// TwinCAT 3 PLC project Untitled1
// ProjectVersion: 1.2.0
// ProgramVersion: 3.1.4023.0
// libraries:
//   Tc2_DataExchange, * (Beckhoff Automation GmbH)
//   Tc2_MC2, * (Beckhoff Automation GmbH)
//   Tc2_SerialCom, * (Beckhoff Automation GmbH)
//   Tc2_Standard, * (Beckhoff Automation GmbH)
//   Tc2_System, * (Beckhoff Automation GmbH)
//   Tc2_Utilities, * (Beckhoff Automation GmbH)
//   Tc3_Module, * (Beckhoff Automation GmbH)
// project tree:
//   DUTs/Communication/Axis/ commAxis.TcDUT
//   DUTs/Communication/ Block128Words.TcDUT, CellDataBlock.TcDUT, commManual.TcDUT, contextVacuum.TcDUT, contextManual.TcDUT
//   DUTs/Communication/Command/ commCommandBase.TcDUT, commCommandGeneric.TcDUT, commCommandPos.TcDUT
//   DUTs/Communication/Cylinder/ commCylinder.TcDUT
//   DUTs/Communication/Signal/ commSignal.TcDUT
//   DUTs/Communication/Unit/ commUnit.TcDUT, commUnitConfig.TcDUT, commUnitGeneric.TcDUT, commUnitController.TcDUT
//   DUTs/Definitions/ eAdsIndexGroups.TcDUT, eCommandTypes.TcDUT, eErrorCodes.TcTLEO, eModes.TcDUT, eCategrories.TcDUT, eCylinderCommands.TcDUT, eErrorClearWays.TcDUT, ePositionType.TcDUT, eOperationModes.TcDUT, eSpecialStates.TcDUT
//   DUTs/HRASI/ defAlignment.TcDUT, defHandshake.TcDUT, defItem.TcDUT, eErrorReasons.TcDUT, eSCARATask.TcTLEO, defSensorPair.TcDUT
//   DUTs/Internal/ ParameterGeneric.TcDUT, ParameterSet.TcDUT, ParametersHome.TcPOU, ParametersPosition.TcDUT
//   DUTs/ ioBundleConveyor.TcDUT, ioBundleET.TcDUT, ioBundleLabelGripper.TcDUT, ioBundlePrinterApplicator.TcDUT
//   DUTs/Material/ MaterialBlock.TcDUT, MaterialHeader.TcDUT
//   GVLs/ GVL.TcGVL, GVL_DeivceList.TcGVL
//   / PlcTask.TcTTO
//   POUs/ CheckBounds.TcPOU, CheckPointer.TcPOU, IncNoOverflow.TcPOU, MAIN.TcPOU
//   POUs/Foundation/ CommonBase.TcPOU, ExecuteBase.TcPOU, InterfaceControlV2.TcPOU, InterfaceManualV2.TcPOU, ProgrammedOutput.TcPOU, RunGroupNode.TcPOU, RunMaterial.TcPOU, RunSafetyFacilityProcessor.TcPOU, RunUnitControllerV2.TcPOU, RunUnitSlave.TcPOU, RunVacuum.TcPOU, SemephoreV1.TcPOU, SemephoreV2.TcPOU, RunAxis.TcPOU, InterfaceControlV1.TcPOU, RunCylinder.TcPOU, InterfaceManualV1.TcPOU, RunSignal.TcPOU, RunUnitControllerV1.TcPOU, RunUnitGeneric.TcPOU, RunUnitIndexerMaster.TcPOU, RunUnitTransporterBase.TcPOU
//   POUs/Helper/ CellDataBlock2Parameter.TcPOU, Parameter2CellDataBlock.TcPOU
//   POUs/Stations/CellularD/ RunCableHolder.TcPOU, RunGradeOutput.TcPOU, RunLabelHandler.TcPOU
//   POUs/Stations/HRASI/InitAndTaskControl/ RunCoordinator.TcPOU, RunInitClamperAndIndexer.TcPOU, RunInitScaraAndRack.TcPOU
//   POUs/Stations/HRASI/ RunBin.TcPOU, RunClamper.TcPOU, RunCommonRack.TcPOU, helperOutputSelection.TcPOU, RunAoiInspectionV1.TcPOU, RunBridge.TcPOU, RunDimmerControl.TcPOU, RunLoading.TcPOU, RunPnueIndexer.TcPOU, RunScaraAgent.TcPOU
//   POUs/Stations/ RunAoiHandshaking.TcPOU (excluded from build), RunAxisAoiView.TcPOU (excluded from build), RunAxisInspection.TcPOU (excluded from build), RunBottomView.TcPOU (excluded from build), RunETest.TcPOU (excluded from build), RunInputV1.TcPOU (excluded from build), RunUnitCellularAIO.TcPOU (excluded from build), RunUnitCellularC.TcPOU (excluded from build), RunLifterCelluar.TcPOU (excluded from build), RunUnitCellularA.TcPOU (excluded from build), RunUnitDummy.TcPOU (excluded from build)
// real-time tasks:
//   TASK PlcTask: cycle T#10ms, priority 20, ADS port 350
// motion (NC):
//   TASK NC-Task 1 SAF: cycle T#2ms, priority 4, ADS port 501
//   TASK NC-Task 1 SVB: cycle T#10ms, priority 8, ADS port 511
//   AXIS Simu1 (id 1)
//     OtherSettings: AllowMotionCmdToSlave=true
//     encoder EncType=1
//     drive DrvType=5
//       Analog: ScaleFactorActTorque=0.1
//       TimeComp: TaskDelayCycles=1
//     controller CtrType=1
//       CtrPara: PriorControlFactor=1
//         Observer: BandWidth=20
//   AXIS Simu2 (id 2)
//     OtherSettings: AllowMotionCmdToSlave=true
//     encoder EncType=1
//     drive DrvType=5
//       Analog: ScaleFactorActTorque=0.1
//       TimeComp: TaskDelayCycles=1
//     controller CtrType=1
//       CtrPara: PriorControlFactor=1
//         Observer: BandWidth=20
//   AXIS Lifter2 (id 3)
//     OtherSettings: AllowMotionCmdToSlave=true
//     encoder EncType=1
//       EncPara: ScaleFactorNumerator=1, ScaleFactorDenominator=8388608
//     drive DrvType=5
//       Analog: ScaleFactorActTorque=0.1
//       TimeComp: TaskDelayCycles=1
//     controller CtrType=1
//       CtrPara: PriorControlFactor=1
//         Observer: BandWidth=20
//   AXIS Lifter3 (id 4)
//     Dynamic: AccelerationMaximum=3500, DecelerationMaximum=3500, Acceleration=3500, Deceleration=3500
//     Velo: SlowManual=10, FastManual=35, Maximum=50
//     OtherSettings: AllowMotionCmdToSlave=true
//     encoder EncType=1
//       EncPara: ScaleFactorNumerator=1, ScaleFactorDenominator=8388608
//     drive DrvType=5
//       Analog: VeloReferenz=50, ScaleFactorActTorque=0.1
//       TimeComp: TaskDelayCycles=1
//     controller CtrType=1
//       CtrPara: PriorControlFactor=1
//         PID: PosKp=50
//         Observer: BandWidth=20
//   AXIS Lifter1 (id 5)
//     OtherSettings: AllowMotionCmdToSlave=true
//     encoder EncType=1
//       EncPara: ScaleFactorNumerator=1, ScaleFactorDenominator=8388608
//     drive DrvType=5
//       Analog: ScaleFactorActTorque=0.1
//       TimeComp: TaskDelayCycles=1
//     controller CtrType=1
//       CtrPara: PriorControlFactor=1
//         Observer: BandWidth=20
//   AXIS Conveyor (id 7)
//     Dynamic: Acceleration=12937.5, Deceleration=12937.5, Jerk=38812.5
//     Velo: RefSearch=86.25, RefSync=86.25, SlowManual=431.25, FastManual=2587.5, Fast=8625, Maximum=8625
//     OtherSettings: AllowMotionCmdToSlave=true
//     encoder EncType=1
//       EncPara: ScaleFactorNumerator=150, ScaleFactorDenominator=1048576, Inverse=true
//     drive DrvType=5
//       DrvPara: Inverse=true
//         Analog: VeloReferenz=9487.5, ScaleFactorActTorque=0.1
//         TimeComp: TaskDelayCycles=1
//     controller CtrType=1
//       CtrPara: PriorControlFactor=1
//         PosDiffControl: Enable=false
//         PID: PosKp=50
//         Observer: BandWidth=20
//   AXIS Horizon1 (id 8)
//     Dynamic: Acceleration=431.25, Deceleration=431.25, Jerk=1293.75
//     Velo: RefSearch=2.875, RefSync=2.875, SlowManual=14.375, FastManual=86.25, Fast=287.5, Maximum=287.5
//     OtherSettings: AllowMotionCmdToSlave=true
//     encoder EncType=1
//       EncPara: ScaleFactorNumerator=5, ScaleFactorDenominator=1048576, Inverse=true
//     drive DrvType=5
//       DrvPara: Inverse=true
//         Analog: VeloReferenz=316.25, ScaleFactorActTorque=0.1
//         TimeComp: TaskDelayCycles=1
//     controller CtrType=1
//       CtrPara: PriorControlFactor=1
//         Observer: BandWidth=20
//   AXIS Horizon2 (id 9)
//     Dynamic: Acceleration=431.25, Deceleration=431.25, Jerk=1293.75
//     Velo: RefSearch=2.875, RefSync=2.875, SlowManual=14.375, FastManual=86.25, Fast=287.5, Maximum=287.5
//     OtherSettings: AllowMotionCmdToSlave=true
//     encoder EncType=1
//       EncPara: ScaleFactorNumerator=5, ScaleFactorDenominator=1048576, Inverse=true
//     drive DrvType=5
//       DrvPara: Inverse=true
//         Analog: VeloReferenz=316.25, ScaleFactorActTorque=0.1
//         TimeComp: TaskDelayCycles=1
//     controller CtrType=1
//       CtrPara: PriorControlFactor=1
//         Observer: BandWidth=20
//   AXIS Horizon3 (id 10)
//     Dynamic: Acceleration=431.25, Deceleration=431.25, Jerk=1293.75
//     Velo: RefSearch=2.875, RefSync=2.875, SlowManual=14.375, FastManual=86.25, Fast=287.5, Maximum=287.5
//     OtherSettings: AllowMotionCmdToSlave=true
//     encoder EncType=1
//       EncPara: ScaleFactorNumerator=5, ScaleFactorDenominator=1048576, Inverse=true
//     drive DrvType=5
//       DrvPara: Inverse=true
//         Analog: VeloReferenz=316.25, ScaleFactorActTorque=0.1
//         TimeComp: TaskDelayCycles=1
//     controller CtrType=1
//       CtrPara: PriorControlFactor=1
//         Observer: BandWidth=20
// I/O:
//   DEVICE Device 1 (EtherCAT) (disabled), AmsNetId 10.221.24.70.2.1
//     Term 1 (EK1200) [EK1200-5000 EtherCAT Power supply (2A E-Bus)]
//       Term 2 (EL1889) [EL1889 16Ch. Dig. Input 24V, 3ms, negative]
//       Term 3 (EL2889) [EL2889 16Ch. Dig. Output 24V, 0.5A, negative]
//       Term 4 (EL6900) [EL6900, TwinSAFE PLC]
//       Term 5 (EL1904) [EL1904, 4 Ch. Safety Input 24V, TwinSAFE]
//         modules: Module 1 (FSOES)
//       Term 6 (EL2904) [EL2904, 4 Ch. Safety Output 24V, 0.5A, TwinSAFE]
//         modules: Module 1 (FSOES), Module 2 (DO)
//       Term 7 (EL9576) [EL9576 Brake chopper terminal]
//       Term 8 (EL7201-9014) [EL7201-9014 1Ch. MDP742 Servo motor output stage with OCT (50V, 2.8A RMS) and STO input]
//       Term 9 (EL7201-9014) [EL7201-9014 1Ch. MDP742 Servo motor output stage with OCT (50V, 2.8A RMS) and STO input]
//       Term 10 (EL7201-9014) [EL7201-9014 1Ch. MDP742 Servo motor output stage with OCT (50V, 2.8A RMS) and STO input]
//       Term 11 (EL7201-9014) [EL7201-9014 1Ch. MDP742 Servo motor output stage with OCT (50V, 2.8A RMS) and STO input]
//       Term 12 (EK1110) [EK1110 EtherCAT extension]
//     Drive 13 (MADLN05BE) [MADLN05BE]
//     Drive 14 (MADLN05BE) [MADLN05BE]
//     Drive 15 (MADLN05BE) [MADLN05BE]
//     Box 16 (NU-EC1) [NU-EC1 (Rev 0004)]

CONFIGURATION Untitled1
    RESOURCE PLC ON TwinCAT3
        TASK PlcTask(INTERVAL := T#10ms, PRIORITY := 20);
        PROGRAM MAIN_D WITH PlcTask : MAIN_D;
    END_RESOURCE
END_CONFIGURATION

// ---- DUTs/Communication/Axis/commAxis.TcDUT
TYPE commAxis :
STRUCT
	operationMonitor :WORD; //0 ,status of servoOn,alarmClear (PLC->HMI
	reserved1 : WORD;//1
	posCommand : DINT; //2-3 , 
	runStatus : DWORD; //4,5 ,  runningWithServoOn , servoReady
	warning : DWORD;//6-7 ,
	alarm: DWORD;//8-9	   ,  64Bits error code
	commandStatus : DWORD; //10,11 , not implemented
	posStatus:WORD;//12,13 , not implemented
	//
	posFeedback : DINT;//14-15
	speedFeedback : DINT;//16-17
	torqueFeedback : DINT;//18-19
	reserved2 : ARRAY[1..4] OF WORD;//20-23
	operationOperation : WORD;//24 , operation of servoOn,alarmClear (HMI->PLC
	reserved3 : ARRAY[1..7] OF WORD; //25-31
	//Depreciated variables suitable for MechtrolinkIII
	address : WORD; //32
	axisType : WORD; //33
	limitPlus : DINT; //34
	limitMinus : DINT; //36
	speedMax : DINT; //38
	positionTolerance : DINT; //40
	boolParameter : WORD; //42 , bit0 , enablePosLimit , bit1 , enableNegLimit
END_STRUCT
END_TYPE

// ---- DUTs/Communication/Block128Words.TcDUT
TYPE Block128Words :
UNION
	reserved : ARRAY[1..128] OF WORD;
	unit : commUnitGeneric;
	material : materialBlock;
END_UNION
END_TYPE

// ---- DUTs/Communication/CellDataBlock.TcDUT
TYPE CellDataBlock :
UNION
	reserved : ARRAY[1..64] OF WORD; //memeory occupation
	axis : commAxis;
	cylinder : commCylinder;
	signal : commSignal;
	command : commCommandGeneric;
	unit : commUnitGeneric;
	//----------
	//	New added , 20191228
	//----------
	vacuum : contextVacuum;
END_UNION
END_TYPE

// ---- DUTs/Communication/Command/commCommandBase.TcDUT
TYPE commCommandBase :
STRUCT	
	axisId: WORD;				//0
	commandType:eCommandTypes;	//1
	speed:DWORD ; // in 0.001mm , fixed point , 2
	accTime:DWORD; // in ms , 4
	decTime:DWORD; // in ms , 6
	torqueLimit:DWORD; // in 0.01 percentage , 8
	subIndex : WORD; //10 , indicate which bank index would be set/read
	reserved : ARRAY[1..5] OF WORD; //11...15
END_STRUCT
END_TYPE

// ---- DUTs/Communication/Command/commCommandGeneric.TcDUT
TYPE commCommandGeneric :
UNION
	base : commCommandBase;
	position : commCommandPos;
END_UNION
END_TYPE

// ---- DUTs/Communication/Command/commCommandPos.TcDUT
TYPE commCommandPos EXTENDS commCommandBase :
STRUCT
	controlWord:DWORD; //16,17 , bit0, true=abs
	coordinate:DINT; //18,19 , in 0.001mm
END_STRUCT
END_TYPE

// ---- DUTs/Communication/commManual.TcDUT
TYPE commManual :
UNION
	comm AT%M* : ARRAY[0..255] OF UINT;
	context : contextManual;
END_UNION
END_TYPE

// ---- DUTs/Communication/contextVacuum.TcDUT
TYPE contextVacuum :
STRUCT
	statusWord : WORD; //0
	command : eCylinderCommands; //1
	lastCommand : eCylinderCommands; //2
	timerCountValue : WORD; //3
	reserved1 : ARRAY[1..4] OF WORD; //4..7
	//context
	threshold : WORD; //8
	vacuumValue : WORD; //9
	reserved3 : ARRAY[1..6] OF WORD; //10-15
	timerSetValue : WORD; //16
	reserved4 : WORD; //17
	//Depre
	reserved5 : WORD; //18
	reserved6 : WORD; //19
END_STRUCT
END_TYPE

// ---- DUTs/Communication/contextManual.TcDUT
TYPE contextManual :
STRUCT
	wordOut  : WORD; //0
		reserved1 : ARRAY[1..31] OF WORD; //1-31
	wordIn	 : WORD; //32
		reserved2 : ARRAY[1..7] OF WORD;  //33-39
	monitorType : eCategrories;//40
	monitorIndex : WORD;//41 , 1-based index
	commitMode : eModes;//42
		reserved3 : WORD; //43
	commitSelection : eCategrories;//44
		reserved4 : WORD; //45
	commitIndex  : WORD;//46 , 1-based index
		reserved5  : ARRAY[1..17] OF WORD; //47-63
	commitBlock  : CellDataBlock;//64
	monitorBlock  : CellDataBlock;//128
END_STRUCT
END_TYPE

// ---- DUTs/Communication/Cylinder/commCylinder.TcDUT
TYPE commCylinder :
STRUCT
	statusWord : WORD; //0
	command : eCylinderCommands; //1
	lastCommand : eCylinderCommands; //2
	timerCountValue : WORD; //3
	reserved1 : ARRAY[1..4] OF WORD; //4..7
	//context
	timerDelayToA : WORD; //8
	timerDelayToB : WORD; //9
	reserved2 : ARRAY[1..6] OF WORD; //10-15
	timerSetValue : WORD; //16
	reserved3 : WORD; //17
	//Depre
	sensorAUsedCount : WORD; //18
	sensorBUsedCount : WORD; //19
END_STRUCT
END_TYPE

// ---- DUTs/Communication/Signal/commSignal.TcDUT
TYPE commSignal :
STRUCT
	address : WORD;	//0
	widthOn : WORD; //1
	widthOff : WORD; //2
	widthOnCount : WORD;//3
	widthOffCount : WORD;//4
	outputWord: WORD;//5
END_STRUCT
END_TYPE

// ---- DUTs/Communication/Unit/commUnit.TcDUT
TYPE commUnit :
	//32Bytes , 16Word occupation
STRUCT
	parent : WORD := 1; //0
	state : WORD;
	alarmCode : WORD;
	
	//Bit0 , enable step control
	//Bit1 , trigger step control
	//Bit2 , pause state
	//Bit3 , (indexer slave) direct off working signal
	//Bit4 , (indexer slave) working signal override
	//Bit5 , (indexer slave) material is valid
	//Bit6 , 
	//Bit7 , last pause parent status
	controlWord : WORD; //3
	//
	nextState : WORD; //4
	serialTransition : BOOL; //5.0
	transitionByte : BYTE; //5.1
	materialBase : WORD; //6
	materialCount : WORD;//7
	//
	reserved1 : DWORD;//8-9
	workingTimerCache : DWORD; //10-11 , used to reflect timer couting
	//
	reservedRest : ARRAY[1..20] OF WORD; //12-31
END_STRUCT
END_TYPE

// ---- DUTs/Communication/Unit/commUnitConfig.TcDUT
TYPE commUnitConfig :
STRUCT
	unitId : WORD; //0
	configId: WORD;//1
	value : DWORD;//2
END_STRUCT
END_TYPE

// ---- DUTs/Communication/Unit/commUnitGeneric.TcDUT
TYPE commUnitGeneric :
UNION
	base : commUnit;
	controller : commUnitController;
	config : commUnitConfig;
	//master : UnitIndexerMaster;
	//slave : UnitIndexerSlave;
END_UNION
END_TYPE

// ---- DUTs/Communication/Unit/commUnitController.TcDUT
TYPE commUnitController EXTENDS commUnit :
STRUCT
	control : DWORD := 16#8; //32
	errorIndex : DWORD; //34
	errorType : DWORD; //36
	//due to memory alignment issue , had to seperate two dword
	errorCode1 : DWORD; // 38
	errorCode2 : DWORD; // 40
	
	reserved2 : ARRAY[42..47] OF WORD; //42-46
	monitorDatas : ARRAY[0..7] OF DWORD; //48-62
END_STRUCT
END_TYPE

// ---- DUTs/Definitions/eAdsIndexGroups.TcDUT
{attribute 'qualified_only'}
{attribute 'strict'}
TYPE eAdsIndexGroups :
(
	RESERVED1 := 16#0,
	RESERVED2 := 16#FFF,
	PLC_ADS_PARA := 16#1000,
	PLC_ADS_STAT := 16#2000,
	PLC_ADS_UNIT := 16#3000,
	//%M fields
	PLCADS_RWM := 16#4020,
	PLCADS_RWMX := 16#4021,
	PLCADS_IGR_RMSIZE := 16#4025,
	PLCADS_IGR_RWRB := 16#4030,
	PLCADS_IGR_RRSIZE := 16#4035,
	PLCADS_IGR_RWDB := 16#4040,
	PLCADS_IGR_RDSIZE := 16#4045,
	//$I,Q fields
	PLCADS_RWI := 16#F020,
	PLCADS_RWQ := 16#F030
);
END_TYPE

// ---- DUTs/Definitions/eCommandTypes.TcDUT
{attribute 'qualified_only'}
{attribute 'strict'}
TYPE eCommandTypes :
(
	NO_OPERATION := 0,
	POSITION:=1,
	ZRET:=3,
	
	SET_POSITION:=16#FF
) WORD;
END_TYPE

// ---- DUTs/Definitions/eErrorCodes.TcTLEO
{attribute 'qualified_only'}
{attribute 'strict'}
TYPE eErrorCodes : 
(
	AC_CONVEYOR_JAMMED := 16#101 , 
	AC_CONVEYOR_NOT_REACHED := 16#102,  
	AC_ET_USAGE_MEET := 16#201,
	AC_ET_SERIES_NG := 16#202
) UDINT;
END_TYPE
//  AC_CONVEYOR_JAMMED = '16#101'
//  AC_CONVEYOR_NOT_REACHED = '16#102'
//  AC_ET_USAGE_MEET = '16#201'
//  AC_ET_SERIES_NG = '16#202'

// ---- DUTs/Definitions/eModes.TcDUT
{attribute 'qualified_only'}
//{attribute 'strict'}
TYPE eModes :
(
	MODE_EXE_AXIS := TO_WORD(eCategrories.SELECTION_AXIS),
    MODE_EXE_CYLINDER := TO_WORD(eCategrories.SELECTION_CYLINDER),
    MODE_EXE_SIGNAL := TO_WORD(eCategrories.SELECTION_SIGNAL), //dummy

    MODE_EXE_COMMAND_BLOCK := TO_WORD(eCategrories.SELECTION_COMMAND_BLOCK),

    MODE_EXE_UNIT := TO_WORD(eCategrories.SELECTION_UNIT),

    MODE_DOWNLOAD_DATA_BLOCK := 15, //PLC<-HMI
    MODE_UPLOAD_DATA_BLOCK := 16,   //PLC->HMI
	
	MODE_EXE_VACUUM := TO_WORD(eCategrories.SELECTION_VACUUM) //new type
) WORD ;
END_TYPE

// ---- DUTs/Definitions/eCategrories.TcDUT
{attribute 'qualified_only'}
{attribute 'strict'}
TYPE eCategrories :
(
	SELECTION_AXIS := 0,
    SELECTION_CYLINDER := 1,
    SELECTION_SIGNAL :=2,
    SELECTION_COMMAND_BLOCK := 4,
    SELECTION_UNIT := 5,
	//-----------
	SELECTION_VACUUM := 6 //add 2019.11.30
) WORD;
END_TYPE

// ---- DUTs/Definitions/eCylinderCommands.TcDUT
{attribute 'qualified_only'}
//{attribute 'strict'}
TYPE eCylinderCommands :
(
	NO_COMMAND := 0,
	COMMAND_A := 1,
	COMMAND_B := 2
) WORD;
END_TYPE

// ---- DUTs/Definitions/eErrorClearWays.TcDUT
{attribute 'qualified_only'}
{attribute 'strict'}
TYPE eErrorClearWays :
(
	NO_ACTION:=0,
	RESET := 1,
	IGNORE :=2
);
END_TYPE

// ---- DUTs/Definitions/ePositionType.TcDUT
{attribute 'qualified_only'}
{attribute 'strict'}
TYPE ePositionType :
(
	POSITION_ABS := 0,
	POSITION_REL := 1
);
END_TYPE

// ---- DUTs/Definitions/eOperationModes.TcDUT
{attribute 'qualified_only'}
{attribute 'strict'}
TYPE eOperationModes :
(
	AUTO := 0, //fully auto
	SEMI_AUTO:=1, //working station trigger...etc
	MANUAL:=2 //axis,cylinder setting/testing
);
END_TYPE

// ---- DUTs/Definitions/eSpecialStates.TcDUT
{attribute 'qualified_only'}
//{attribute 'strict'}
TYPE eSpecialStates : 
(
	INITIAL_BEGIN := 16#100,
	INITIAL_STATE_1 := INITIAL_BEGIN+1,
	INITIAL_STATE_2 := INITIAL_BEGIN+2,
	INITIAL_STATE_3 := INITIAL_BEGIN+3,
	INITIAL_STATE_4 := INITIAL_BEGIN+4,
	INITIAL_STATE_5 := INITIAL_BEGIN+5,
	INITIAL_STATE_6 := INITIAL_BEGIN+6,
	INITIAL_STATE_7 := INITIAL_BEGIN+7,
	INITIAL_END := 16#1FF, //256 states possible
	INITIAL_REGION := 16#F00,
	
	SLAVE_WORK_TRIGGER := 16#0,
	SLAVE_ENTER_PROCEDURE := 16#200,
	SLAVE_WORK_DONE := 16#FF,
	
	SLAVE_AXIS_INSPECTION_ENTER := 16#300, //enter iteration region
	SLAVE_AXIS_INSPECTION_ITERATION := 16#301,
	SLAVE_AXIS_INSPECTION_EXIT := 16#400, //exit iteration region
	
	GENERIC_GROUP_START := 0, //working sequence start , but need to skip interval of initial region
	GENERIC_GROUP_IDLE := 16#1,
	//
	MAIN_WAIT_INITIALIZING := 16#800,
	MAIN_INITIALIZING := 16#801,
	MAIN_INITIALIZED := 16#802,	
	
	FORBIDDEN := 16#FFFF
) INT ;
END_TYPE

// ---- DUTs/HRASI/defAlignment.TcDUT
TYPE defAlignment :
STRUCT
	//-----------------
	//	Input from I/O
	//-----------------	
	ioJobComplete AT%I*:BOOL;
	ioAcqComplete AT%I*:BOOL;
	//-----------------
	//	Output to I/O
	//-----------------	
	ioTrigger AT%Q*:BOOL;
	//-----------------
	//	Input from SCARA
	//-----------------
	alignTrigger AT%I*: BOOL;
	alignSelection AT%I*: BYTE;
	//-----------------
	//	Output to SCARA
	//-----------------
	alignJobComplete AT%Q*: BOOL;
	alignAcqComplete AT%Q*: BOOL;
	
	alignX AT%Q*: REAL;
	alignY AT%Q*: REAL;
	alignU AT%Q*: REAL;
END_STRUCT
END_TYPE

// ---- DUTs/HRASI/defHandshake.TcDUT
TYPE defHandshake :
STRUCT
	ready AT%Q* : BOOL;
	ack AT%I*: BOOL;
	
	valid AT%I*: BOOL; // whether material presented after work done
END_STRUCT
END_TYPE

// ---- DUTs/HRASI/defItem.TcDUT
TYPE defItem :
STRUCT
	CurrerntIndex AT%I* : BYTE; //curent working index
	Counter AT%I* : BYTE;  //successful picked item amount	
	Bound : BYTE;
END_STRUCT
END_TYPE

// ---- DUTs/HRASI/eErrorReasons.TcDUT
{attribute 'qualified_only'}
{attribute 'strict'}
TYPE eErrorReasons :
(
	ERR_NOR:=0,
	ERR_PART_REMAINED:=400,
	ERR_PART_MISSING:=401,
	ERR_CONSECUTIVE_NG:=8001,
	ERR_TOP_MISPLACED:=8000,
	ERR_BOTTOM_UP_SIDE_DOWN:=8002,
	ERR_USER_ACK:=8010,
	ERR_GENERIC_ERROR:=8500,
	ERR_SYSTEM_ERROR:=4000,
	ERR_IDLE:=500,
	ERR_OFFLINE:=501,
	ERR_EMG:=1,
	ERR_INCORRECT_AIR:=10,
	ERR_SAFETY:=8501,
	ERR_VACUUM_JAMMED:=600
) DWORD;
END_TYPE

// ---- DUTs/HRASI/eSCARATask.TcTLEO
{attribute 'qualified_only'}
{attribute 'strict'}
TYPE eSCARATask :
(
	task_init := 0,
	task_regular_check_scara1 := 1,
	task_regular_check_scara2 := 2,
	task_assemble_scara1 := 3,
	task_snap_scara2 := 4,
	task_load_drop :=5
) INT;
END_TYPE

// ---- DUTs/HRASI/defSensorPair.TcDUT
TYPE defSensorPair :
STRUCT
	bit0 AT%I* : BOOL;
	bit1 AT%I* : BOOL;
END_STRUCT
END_TYPE

// ---- DUTs/Internal/ParameterGeneric.TcDUT
TYPE ParameterGeneric :
UNION
	position : ParametersPosition;
	home : ParametersHome;
END_UNION
END_TYPE

// ---- DUTs/Internal/ParameterSet.TcDUT
TYPE ParameterSet :
STRUCT
	command : eCommandTypes := eCommandTypes.POSITION;
	parameter : ParameterGeneric;
END_STRUCT
END_TYPE

// ---- DUTs/Internal/ParametersPosition.TcDUT
TYPE ParametersPosition :
STRUCT
	Velocity : LREAL := 10; //in mm/s
	Acceleration: LREAL := 100; // in mm/s2
	Deceleration: LREAL := 100;
	Position: LREAL := 10; // in mm
	PositionType : ePositionType := ePositionType.POSITION_ABS;
END_STRUCT
END_TYPE

// ---- DUTs/ioBundleConveyor.TcDUT
TYPE ioBundleConveyor :
STRUCT
	overheat AT%I* : BIT;
	run AT%Q* : BIT;
END_STRUCT
END_TYPE

// ---- DUTs/ioBundleET.TcDUT
TYPE ioBundleET :
STRUCT
	external AT%Q* : BIT;
	hipot AT%Q* : BIT;
	i1 AT%Q* : BIT;
	i2 AT%Q* : BIT;
	
	o1 AT%I* : BIT;
	o2 AT%I* : BIT;
	o3 AT%I* : BIT; //pin7, attached
	o4 AT%I* : BIT; //pin8, OK/NG
	o5 AT%I* : BIT;
	o6 at%I* : BIT;

END_STRUCT
END_TYPE

// ---- DUTs/ioBundleLabelGripper.TcDUT
TYPE ioBundleLabelGripper :
STRUCT
	vacuumGripper AT%Q* : BIT;
	breakGripper AT%Q* : BIT;
	
	vacuumPressor AT%Q* : BIT;
	breakPressor AT%Q* : BIT;
	
END_STRUCT
END_TYPE

// ---- DUTs/ioBundlePrinterApplicator.TcDUT
TYPE ioBundlePrinterApplicator :
STRUCT
	prtStart AT%Q* : BIT;
	prtFeed AT%Q* : BIT;
	prtPause AT%Q* : BIT;
	prtReprint AT%Q* : BIT;
	
	prtRiblow AT%I* : BIT;
	prtSerReq AT%I* : BIT;
	prtEnd AT%I* : BIT;
	prtPrtMout AT%I* : BIT;
	prtRibout AT%I* : BIT;
	prtData AT%I* : BIT;
END_STRUCT
END_TYPE

// ---- DUTs/Material/MaterialBlock.TcDUT
TYPE MaterialBlock :
STRUCT
	data : ARRAY[0..63] OF WORD;
END_STRUCT
END_TYPE

// ---- DUTs/Material/MaterialHeader.TcDUT
TYPE MaterialHeader :
STRUCT
	wordOut : WORD; //0, bit1:Act,bit2:IsValid,bit3:schedualed
		reserved1 : ARRAY[1..7] OF WORD; //1-7
	wordIn : WORD;//8 , 2,Done,bit0:engaged,bit1:done
		reserved2 : ARRAY[9..15] OF WORD; //9-15
	
	id : DWORD;//16 , 32bits
	
		reserved3 : ARRAY[1..2] of word;//18-19
	//Protocal ver2 , Act on->Act off
END_STRUCT
END_TYPE

// ---- GVLs/GVL.TcGVL
{attribute 'qualified_only'}
VAR_GLOBAL
	//
	ioConveyor : ioBundleConveyor;
	ioControl : ioBundleControl;
	ioSafety : ioBundleSafety;
	ioPrinter : ioBundlePrinterApplicator;
	ioLabelHandler : ioBundleLabelGripper;

	cylinderControls : ARRAY[1..16] OF RunCylinder;
	signalControls : ARRAY[1..10] OF RunSignal;
	axisControls: ARRAY[1..5] OF RunAxis;
	//
	materialSlots AT%M* : ARRAY[1..4] OF Block128Words;	
	stations : ARRAY[1..8] OF POINTER TO RunUnitGeneric;
		
	//for downstream
	//downstreamSyncEngaged AT%MB127 : BOOL;
	//downstreamSyncAcknowledged AT%MB128 : BOOL;
	
	bObjectsLinked : BOOL;
END_VAR

// ---- GVLs/GVL_DeivceList.TcGVL
//{attribute 'qualified_only'}
VAR_GLOBAL
	//-------
	//Signals
	//-------
	A19: INT :=1; //Bottom upside-down check
	A23: INT :=2; //Product bin
	A24: INT :=3; //NG bin
	A25: INT :=4; //FQC bin
	B18: INT :=5; //Empty nest
	B19: INT :=6; //S/V Check#1
	B21: INT :=7; //Rack1 Approach
	B22: INT :=8; //Rack3 Approach
	B25: INT :=9; //Rack2 Approach
	B26: INT :=10; //Rack4 Approach

	S2: INT :=11; //START
	S3: INT :=12; //STOP
	S4: INT :=13; //RESET
	S5: INT :=14; //DOOR UNLOCK
	S6: INT :=15; //RACK1
	S7: INT :=16; //RACK2
	S8: INT :=17; //RACK3
	S9: INT :=18; //RACK4
	//--------------
	//Cylinders
	//--------------
	Cy1: INT :=1; //Filter#1 vertical cylinder
	Cy10: INT :=2; //Rack3
	Cy11: INT :=3; //Rack4
	Cy12: INT :=4; //Clamper axial#A
	Cy13: INT :=5; //Clamper hold#A
	Cy14: INT :=6; //Clamper axial#B
	Cy15: INT :=7; //Clamper hold#B
	Cy16: INT :=8; //AOI NG ejector
	Cy17: INT :=9; //Index piston
	Cy18: INT :=10; //Index locker
	Cy2: INT :=11; //Filter#2 vertical cylinder
	Cy3: INT :=12; //Filter#3 vertical cylinder
	Cy6: INT :=13; //Top part holder
	Cy7: INT :=14; //Bottom part vertical
	Cy8: INT :=15; //Rack1
	Cy9: INT :=16; //Rack2
	//--------------
	//Vacuums
	//--------------
	A10: INT :=1; //Filter#2 vacuum sensor
	A11: INT :=2; //Filter#3-1 vacuum sensor
	A12: INT :=3; //Filter#3-2 vacuum sensor
	A13: INT :=4; //Back secure#1
	A14: INT :=5; //Back secure#2
	A20: INT :=6; //Bottom vacuum check
	A9: INT :=7; //Filter#1 vacuum sensor
	VG1: INT :=8; //Filter#1 rib secure#A
	VG2: INT :=9; //Filter#2 rib secure#A
	VG3: INT :=10; //Filter#3 rib secure#A
	VG4: INT :=11; //Filter#1 rib secure#B
	VG5: INT :=12; //Filter#2 rib secure#B
	VG6: INT :=13; //Filter#3 rib secure#B

	//--------------
	//Material slots
	//--------------
	materialA1 : INT :=1;
	materialA2 : INT :=2;
	materialA3 : INT :=3;
	materialA4 : INT :=4;
END_VAR

// ---- POUs/Foundation/RunCylinder.TcPOU
FUNCTION_BLOCK RunCylinder Extends ExecuteBase
VAR			

	COMMAND_CACHED : eCylinderCommands; //1 , HMI->PLC
	LAST_COMMAND : eCylinderCommands;   //2 , 
		
	ACT_A AT %Q* : ARRAY[1..2] OF BOOL;
	ACT_B AT %Q* : ARRAY[1..2] OF BOOL;
	
	SENSOR_A AT %I* : ARRAY[1..4] OF BOOL;
	SENSOR_B AT %I* : ARRAY[1..4] OF BOOL;

	nCounter : INT := 0;
	bMatched : BOOL := false;
		
	BIT_WARNING : BIT; //0
	BIT_A_MATCH : BIT; //1
	BIT_B_MATCH : BIT; //2
	BIT_WARN_SUPPRESS : BIT; //3 , (Control)
	
	BIT_DONE : BIT; //5
	
	isMatched : BOOL;
	isStrokeReach : BOOL;
END_VAR
VAR PERSISTENT
	A_SENSOR_USED_COUNT : INT := 0;
	B_SENSOR_USED_COUNT : INT :=0 ;		

	TMR_WATCH_DOG : TON ; //Watch dog timer
	TMR_DELAY_TO_A : TON;
	TMR_DELAY_TO_B : TON;
END_VAR

SUPER^();

//Run timers
TMR_WATCH_DOG(IN:= , PT:= , Q=> , ET=> );
TMR_DELAY_TO_A(IN:= , PT:= , Q=> , ET=> );
TMR_DELAY_TO_B(IN:= , PT:= , Q=> , ET=> );

// scan all sensor status
BIT_A_MATCH := TRUE;
FOR nCounter := 1 TO A_SENSOR_USED_COUNT BY 1 DO
	BIT_A_MATCH := (BIT_A_MATCH AND SENSOR_A[nCounter]);
END_FOR
BIT_B_MATCH := TRUE;
FOR nCounter := 1 TO B_SENSOR_USED_COUNT BY 1 DO
	BIT_B_MATCH := (BIT_B_MATCH AND SENSOR_B[nCounter]);
END_FOR

// once command changes , reset timer counter
IF COMMAND_CACHED <> LAST_COMMAND THEN
	TMR_DELAY_TO_A.IN := (COMMAND_CACHED=eCylinderCommands.COMMAND_A); //active A delay timer
	TMR_DELAY_TO_B.IN := (COMMAND_CACHED=eCylinderCommands.COMMAND_B); //if no sensor B , active B delay timer
	
	//reset done/warn
	BIT_DONE := FALSE;
	BIT_WARNING := FALSE;
	
	//output process , for nuetual command , hold current position
	IF COMMAND_CACHED <> eCylinderCommands.NO_COMMAND THEN
		FOR nCounter:=1 TO 2 BY 1 DO
			ACT_A[nCounter] := (COMMAND_CACHED = eCylinderCommands.COMMAND_A);
			ACT_B[nCounter] := (COMMAND_CACHED = eCylinderCommands.COMMAND_B);
		END_FOR
	END_IF
	
END_IF


//reset
bMatched := FALSE;
// Check if match
CASE COMMAND_CACHED OF
	eCylinderCommands.NO_COMMAND:
		bMatched:= TRUE;
	
	eCylinderCommands.COMMAND_A:
	//IF TMR_DELAY_TO_A.Q THEN
		bMatched:= (BIT_A_MATCH OR (A_SENSOR_USED_COUNT=0)) AND ((NOT BIT_B_MATCH) OR (B_SENSOR_USED_COUNT=0));
	//END_IF
	
	eCylinderCommands.COMMAND_B:
	//IF TMR_DELAY_TO_B.Q THEN
		bMatched:= ((NOT BIT_A_MATCH) OR (A_SENSOR_USED_COUNT=0)) AND (BIT_B_MATCH OR (B_SENSOR_USED_COUNT=0) );
	//END_IF
		
END_CASE

//start
IF NOT bMatched AND (TMR_DELAY_TO_B.Q OR TMR_DELAY_TO_A.Q) THEN
	TMR_WATCH_DOG.in := TRUE;
ELSE
	TMR_WATCH_DOG.in := FALSE;
END_IF

// status update
//BIT_DONE :=  isShutVerification OR bMatched OR (NOT bMatched AND (BIT_WARN_SUPPRESS ) AND TMR_WATCH_DOG.Q);
//BIT_WARNING := NOT isShutVerification AND(NOT bMatched) AND (NOT BIT_WARN_SUPPRESS) AND TMR_WATCH_DOG.Q AND (TMR_DELAY_TO_B.Q OR TMR_DELAY_TO_A.Q);

isMatched := bMatched OR (NOT bMatched AND BIT_WARN_SUPPRESS );
isStrokeReach := (TMR_DELAY_TO_B.Q AND COMMAND_CACHED=eCylinderCommands.COMMAND_B) OR  (TMR_DELAY_TO_A.Q AND COMMAND_CACHED=eCylinderCommands.COMMAND_A) OR COMMAND_CACHED=eCylinderCommands.NO_COMMAND;

BIT_DONE :=  isShutVerification OR (isMatched AND isStrokeReach);
BIT_WARNING := NOT isShutVerification AND NOT isMatched AND TMR_WATCH_DOG.Q ;

// cache last command
LAST_COMMAND := COMMAND_CACHED;

//scan-out status
//comm.STATUS_WORD.0 := BIT_WARNING;
//comm.STATUS_WORD.1 := BIT_A_MATCH;
//comm.STATUS_WORD.2 := BIT_B_MATCH;
//comm.STATUS_WORD.5 := BIT_DONE;

METHOD ConfigureRead : CellDataBlock
VAR_INPUT
	input : CellDataBlock; //would offer sub-index ...etc
	mode : eModes;
END_VAR

//ConfigureRead.cylinder.sensorAUsedCount := TO_WORD(A_SENSOR_USED_COUNT);
//ConfigureRead.cylinder.sensorBUsedCount := TO_WORD(B_SENSOR_USED_COUNT);

ConfigureRead.cylinder.timerSetValue := TO_WORD(TMR_WATCH_DOG.PT);
ConfigureRead.cylinder.timerSetValue := TO_WORD(TMR_DELAY_TO_A.PT);
ConfigureRead.cylinder.timerSetValue := TO_WORD(TMR_DELAY_TO_B.PT);
END_METHOD

METHOD ConfigureWrite : BOOL
VAR_INPUT
	input : CellDataBlock;
	mode : eModes;
END_VAR
//A_SENSOR_USED_COUNT := TO_INT(input.cylinder.sensorAUsedCount);
//B_SENSOR_USED_COUNT := TO_INT(input.cylinder.sensorBUsedCount);

TMR_WATCH_DOG.PT := TO_TIME(input.cylinder.timerSetValue);
TMR_DELAY_TO_A.PT := TO_TIME(input.cylinder.timerSetValue);
TMR_DELAY_TO_B.PT := TO_TIME(input.cylinder.timerSetValue);
END_METHOD

METHOD Control : BOOL
VAR_INPUT
	input : CellDataBlock;
	mode : eModes;
END_VAR
Execute(argCommand:= input.cylinder.command);
Control:=true;
END_METHOD

METHOD ErrorClear : BOOL
VAR_INPUT
	input : eErrorClearWays;
END_VAR
CASE input OF
	eErrorClearWays.RESET:
		//Timer reset only
	eErrorClearWays.IGNORE:
		//suppress warning
		BIT_WARN_SUPPRESS := TRUE;
END_CASE
END_METHOD

METHOD ErrorDetect : UDINT
VAR_INPUT
END_VAR
ErrorDetect := 0;
IF BIT_WARNING AND NOT isShutAlarm THEN
	ErrorDetect := COMMAND_CACHED; //distinguish different error 
END_IF
END_METHOD

METHOD Execute : BOOL
VAR_INPUT
	argCommand : eCylinderCommands;
END_VAR
VAR
	outDone  : BOOL ;
END_VAR
// store command
COMMAND_CACHED := argCommand;

outDone := BIT_DONE AND NOT BIT_WARNING AND (COMMAND_CACHED = LAST_COMMAND);

//reset surpress
IF outDone THEN
	BIT_WARN_SUPPRESS := FALSE;
END_IF

Execute:=outDone; //return
END_METHOD

METHOD FB_init : BOOL
VAR_INPUT
	bInitRetains : BOOL; // if TRUE, the retain variables are initialized (warm start / cold start)
	bInCopyCode : BOOL;  // if TRUE, the instance afterwards gets moved into the copy code (online change)
	
	//argASensorUsed : INT := 0;
	//argBSensorUsed : INT := 0;
END_VAR
//A_SENSOR_USED_COUNT := argASensorUsed;
//B_SENSOR_USED_COUNT := argBSensorUsed;

//given timer initial value
//TMR_WATCH_DOG.PT := T#200MS;
//TMR_DELAY_TO_A.PT := T#200MS;
//TMR_DELAY_TO_B.PT := T#200MS;
IF bInitRetains THEN
	TMR_WATCH_DOG.PT := T#200MS;
	TMR_DELAY_TO_A.PT := T#200MS;
	TMR_DELAY_TO_B.PT := T#200MS;
END_IF
END_METHOD

METHOD Monitor : CellDataBlock
VAR_INPUT
END_VAR
VAR CONSTANT
	bit0Warn : INT :=0;
	bit1MonGroupA : INT :=1;
	bit2MonGroupB : INT :=2;
	bit3CtlSuppress : INT :=3;
	bit4TmrOn : INT :=4;
	bit5Done : INT := 5;
	//New
	bit6TmrAOn : INT :=6;
	bit7TmrBOn : INT :=7;
END_VAR
Monitor.cylinder.statusWord.bit0Warn := BIT_WARNING;
Monitor.cylinder.statusWord.bit1MonGroupA := BIT_A_MATCH;
Monitor.cylinder.statusWord.bit2MonGroupB := BIT_B_MATCH;
Monitor.cylinder.statusWord.bit3CtlSuppress := BIT_WARN_SUPPRESS;
Monitor.cylinder.statusWord.bit4TmrOn := TMR_WATCH_DOG.Q;
Monitor.cylinder.statusWord.bit5Done := BIT_DONE;

Monitor.cylinder.statusWord.bit6TmrAOn := TMR_DELAY_TO_A.Q;
Monitor.cylinder.statusWord.bit7TmrBOn := TMR_DELAY_TO_B.Q;

Monitor.cylinder.lastCommand := LAST_COMMAND;
END_METHOD

METHOD TypeCode : eCategrories
VAR_INPUT
END_VAR
TypeCode := eCategrories.SELECTION_CYLINDER;
END_METHOD

END_FUNCTION_BLOCK

// ---- POUs/Foundation/ExecuteBase.TcPOU
FUNCTION_BLOCK ExecuteBase EXTENDS CommonBase
VAR_INPUT
	isRemoteControl : BOOL;
	isShutVerification  : BOOL; //shut verification
	isShutAlarm : bool; //no alarm even warning
END_VAR
VAR_OUTPUT
END_VAR
VAR
	remoteCommand AT%I* : BYTE;
	remoteAcknowledge AT%Q*: BYTE;
	
	internalCommand : eCylinderCommands;
END_VAR

IF isRemoteControl THEN
	IF Execute(argCommand := BYTE_TO_WORD(remoteCommand)) THEN
		remoteAcknowledge := remoteCommand;
	ELSE
		remoteAcknowledge := 0;
	END_IF
END_IF

METHOD Execute : BOOL
VAR_INPUT
	argCommand : eCylinderCommands;
END_VAR
END_METHOD

END_FUNCTION_BLOCK

// ---- POUs/Foundation/CommonBase.TcPOU
FUNCTION_BLOCK CommonBase
VAR_INPUT
END_VAR
VAR_OUTPUT
END_VAR
VAR
	default : INT := 16#FF; //for base class , minimun requires one field to locate address
END_VAR

METHOD ConfigureRead : CellDataBlock
VAR_INPUT
	input : CellDataBlock; //would offer sub-index ...etc
	mode : eModes;
END_VAR
END_METHOD

METHOD ConfigureWrite : BOOL
VAR_INPUT
	input : CellDataBlock;
	mode : eModes;
END_VAR
END_METHOD

METHOD Control : BOOL
VAR_INPUT
	input : CellDataBlock;
	mode : eModes;
END_VAR
END_METHOD

METHOD ErrorClear : BOOL
VAR_INPUT
	input : eErrorClearWays;
END_VAR
END_METHOD

METHOD ErrorDetect : UDINT
VAR_INPUT
END_VAR
END_METHOD

METHOD Monitor : CellDataBlock
VAR_INPUT
END_VAR
END_METHOD

METHOD Stop : BOOL
VAR_INPUT
END_VAR
END_METHOD

METHOD TypeCode : eCategrories
VAR_INPUT
END_VAR
END_METHOD

END_FUNCTION_BLOCK

// ---- POUs/Foundation/RunSignal.TcPOU
FUNCTION_BLOCK RunSignal Extends CommonBase
VAR_INPUT
END_VAR
VAR_OUTPUT
	raw : BOOL;
	debouncedOn AT%Q* : BOOL;
	debouncedOff AT%Q* : BOOL;
	
	onTimeElapsed : TIME;
	offTimeElapsed : TIME;
END_VAR
VAR
	input AT%I* : BOOL;
END_VAR
VAR PERSISTENT
	debouncedOnTimer : TON;
	debouncedOffTimer : TOn;
	
END_VAR


raw := input;

debouncedOnTimer(IN:= input, PT:= , Q=> debouncedOn, ET=> );
debouncedOffTimer(IN:= NOT input, PT:= , Q=> debouncedoff, ET=> );

onTimeElapsed := debouncedOnTimer.ET;
offTimeElapsed := debouncedOffTimer.ET;

METHOD ConfigureRead : CellDataBlock
VAR_INPUT
	input : CellDataBlock; //would offer sub-index ...etc
	mode : eModes;
END_VAR
ConfigureRead.signal.widthOn := TO_WORD(debouncedOnTimer.PT);
ConfigureRead.signal.widthOff := TO_WORD(debouncedOffTimer.PT);
END_METHOD

METHOD ConfigureWrite : BOOL
VAR_INPUT
	input : CellDataBlock;
	mode : eModes;
END_VAR
debouncedOffTimer.PT := TO_TIME(input.signal.widthOff);
debouncedOnTimer.PT := TO_TIME(input.signal.widthOn);
END_METHOD

METHOD FB_init : BOOL
VAR_INPUT
	bInitRetains : BOOL; // if TRUE, the retain variables are initialized (warm start / cold start)
	bInCopyCode : BOOL;  // if TRUE, the instance afterwards gets moved into the copy code (online change)
END_VAR
IF bInitRetains THEN
	debouncedOnTimer.PT := T#100MS;
	debouncedOffTimer.PT := T#100ms;
END_IF
END_METHOD

METHOD Monitor : CellDataBlock
VAR_INPUT
END_VAR
VAR CONSTANT
	indexDebouncedOn : INT := 0;
	indexDebouncedOff : INT := 1;
	indexRaw : INT := 2;
END_VAR
Monitor.signal.widthOffCount := TO_WORD(debouncedOffTimer.ET);
Monitor.signal.widthOnCount := TO_WORD(debouncedOnTimer.ET);

Monitor.signal.outputWord.indexDebouncedOn := debouncedOn;
Monitor.signal.outputWord.indexDebouncedOff := debouncedOff;
Monitor.signal.outputWord.indexRaw := raw;
END_METHOD

END_FUNCTION_BLOCK

// ---- POUs/Foundation/RunAxis.TcPOU
FUNCTION_BLOCK RunAxis EXTENDS CommonBase
VAR_OUTPUT
	PositionFeedback : LREAL;
	//PositionCommand : LREAL;
END_VAR
VAR	
	Axis : AXIS_REF;
	 
	nCounter : int :=0;
	fbMoveAbs : ARRAY[1..3] OF MC_MoveAbsolute; //preset n buffers available
	fbMoveHome : MC_Home;
	fbPower : MC_Power;
	fbReset: MC_Reset;
	fbSetPosition: MC_SetPosition;
	fbStop : MC_Stop;
	
	//Status reading
	fbReadActualVelocity: MC_ReadParameter;
	fbReadActualPosition : MC_ReadActualPosition;
	fbReadCommandPosition : MC_ReadParameter;
	fbReadStatus : MC_ReadStatus;
	fbReadControlOutput : MC_ReadParameter;
	//Parameter writing
	fbWriteLimitPositive : MC_WriteParameterPersistent;
	fbWriteLimitNegtive : MC_WriteParameterPersistent;
	fbEnableLimitPositive : MC_WriteBoolParameter;
	fbEnableLimitNegtive : MC_WriteBoolParameter;
	
	timerFbReset : TON;
	//bMonitoring : bool;
END_VAR
VAR PERSISTENT
	ptpCommands : ARRAY[1..12] OF ParameterSet; //collect command blocks relative to this axis here
	moveAbsCount : INT := 1;
END_VAR
VAR CONSTANT
	typeCode : eCategrories := eCategrories.SELECTION_AXIS;
END_VAR

//----------------------------SW Limit
fbWriteLimitPositive(
	Axis:= Axis, 
	Execute:= , 
	ParameterNumber:= SWLimitPos, 
	Value:= , 
	Done=> , 
	Busy=> , 
	Error=> , 
	ErrorID=> );
IF fbWriteLimitPositive.Execute AND (fbWriteLimitPositive.Done OR fbWriteLimitPositive.Error) THEN
	fbWriteLimitPositive.Execute := FALSE; //auto reset
END_IF
fbWriteLimitNegtive(
	Axis:= Axis, 
	Execute:= , 
	ParameterNumber:= SWLimitNeg, 
	Value:= , 
	Done=> , 
	Busy=> , 
	Error=> , 
	ErrorID=> );
IF fbWriteLimitNegtive.Execute AND (fbWriteLimitNegtive.Done OR fbWriteLimitNegtive.Error) THEN
	fbWriteLimitNegtive.Execute := FALSE;
END_IF
fbEnableLimitPositive(
	Axis:= Axis , 
	Execute:= , 
	ParameterNumber:= EnableLimitPos, 
	Value:= , 
	Done=> , 
	Busy=> , 
	Error=> , 
	ErrorID=> );
IF fbEnableLimitPositive.Execute AND (fbEnableLimitPositive.Done OR fbEnableLimitPositive.Error) THEN
	fbEnableLimitPositive.Execute := FALSE;
END_IF
fbEnableLimitNegtive(
	Axis:= Axis , 
	Execute:= , 
	ParameterNumber:= EnableLimitNeg, 
	Value:= , 
	Done=> , 
	Busy=> , 
	Error=> , 
	ErrorID=> );
IF fbEnableLimitNegtive.Execute AND (fbEnableLimitNegtive.Done OR fbEnableLimitNegtive.Error) THEN
	fbEnableLimitNegtive.Execute := false;
END_IF
//----------------------------

fbReadCommandPosition(
	Axis:= Axis, 
	Enable:= TRUE, 
	ParameterNumber:= CommandedPosition, 
	ReadMode:= READMODE_CYCLIC, 
	Valid=> , 
	Busy=> , 
	Error=> , 
	ErrorID=> , 
	Value=> );


fbSetPosition(
	Axis:= Axis, 
	Execute:= , 
	Position:= , 
	Mode:= , 
	Options:= , 
	Done=> , 
	Busy=> , 
	Error=> , 
	ErrorID=> );

//default mode
fbPower(
	Axis:= Axis, 
	Enable:= , 
	Enable_Positive:= , 
	Enable_Negative:= , 
	Override:= , 
	BufferMode:= , 
	Options:= , 
	Status=> , 
	Busy=> , 
	Active=> , 
	Error=> , 
	ErrorID=> );
	
fbReset(
	Axis:= Axis, 
	Execute:= , 
	Done=> , 
	Busy=> , 
	Error=> , 
	ErrorID=> );

// Reset alarm clear after 100ms
timerFbReset(IN:= fbReset.Execute, PT:= T#100MS, Q=> , ET=> );	
IF timerFbReset.Q THEN
	fbReset.Execute := FALSE;
END_IF
	
//Status reading and update
fbReadActualVelocity(
	Axis:= Axis, 
	Enable:= TRUE, 
	ParameterNumber:= ActualVelocity, 
	ReadMode:= READMODE_CYCLIC, 
	Valid=> , 
	Busy=> , 
	Error=> , 
	ErrorID=> , 
	Value=> );

fbReadActualPosition(
	Axis:= axis, 
	Enable:= TRUE, 
	Valid=> , 
	Busy=> , 
	Error=> , 
	ErrorID=> , 
	Position=> PositionFeedback);
fbReadControlOutput(
	Axis:= axis, 
	Enable:= TRUE, 
	ParameterNumber:= AxisDriveMaxOutputLimitation, 
	ReadMode:= READMODE_CYCLIC, 
	Valid=> , 
	Busy=> , 
	Error=> , 
	ErrorID=> , 
	Value=> );
	
fbReadStatus(
	Axis:= axis, 
	Enable:= TRUE, 
	Valid=> , 
	Busy=> , 
	Error=> , 
	ErrorID=> , 
	ErrorStop=> , 
	Disabled=> , 
	Stopping=> , 
	StandStill=> , 
	DiscreteMotion=> , 
	ContinuousMotion=> , 
	SynchronizedMotion=> , 
	Homing=> , 
	ConstantVelocity=> , 
	Accelerating=> , 
	Decelerating=> , 
	Status=> );
	
fbStop(
	Axis:= Axis, 
	Execute:= , 
	Deceleration:= , 
	Jerk:= , 
	Options:= , 
	Done=> , 
	Busy=> , 
	Active=> , 
	CommandAborted=> , 
	Error=> , 
	ErrorID=> );
	
	
//Reset after cylic
IF fbStop.Execute THEN
	fbStop.Execute := FALSE;
END_IF
	
IF NOT fbPower.Enable THEN
	RETURN; //do not execute following commands
END_IF
	//execute founction blocks once powered
	//possible to configure how many buffer used
	FOR nCounter:=1 TO moveAbsCount BY 1 DO
	fbMoveAbs[nCounter](
		Axis:= Axis, 
		Execute:= , 
		Position:= , 
		Velocity:= , 
		Acceleration:= , 
		Deceleration:= , 
		Jerk:= , 
		BufferMode:= MC_BlendingPrevious, 
		Options:= , 
		Done=> , 
		Busy=> , 
		Active=> , 
		CommandAborted=> , 
		Error=> , 
		ErrorID=> );
	END_FOR
	
		
	fbMoveHome(
		Axis:= Axis, 
		Execute:= , 
		Position:= , 
		HomingMode:= , 
		BufferMode:= , 
		Options:= , 
		bCalibrationCam:= , 
		Done=> , 
		Busy=> , 
		Active=> , 
		CommandAborted=> , 
		Error=> , 
		ErrorID=> );

METHOD ConfigureRead : CellDataBlock
VAR_INPUT
	input : CellDataBlock; //would offer sub-index ...etc
	mode : eModes;
END_VAR
VAR
	temp : ParameterSet; 
END_VAR
VAR CONSTANT
	indexEnablePosLimit : INT := 0;
	indexEnableNegLimit : INT := 0;
END_VAR
CASE mode OF
	eModes.MODE_EXE_AXIS:
		//software limit
		ConfigureRead.axis.limitPlus := TO_DINT(fbWriteLimitPositive.Value / 0.001); 
		ConfigureRead.axis.limitMinus := TO_DINT(fbWriteLimitNegtive.Value / 0.001);
		ConfigureRead.axis.boolParameter.indexEnablePosLimit := fbEnableLimitPositive.Value;
		ConfigureRead.axis.boolParameter.indexEnableNegLimit := fbEnableLimitNegtive.Value  ;
	eModes.MODE_EXE_COMMAND_BLOCK:
		temp := ptpCommands[input.command.base.subIndex+1] ; //write-in
		ConfigureRead := Parameter2CellDataBlock(input:= temp);
		
END_CASE
END_METHOD

METHOD ConfigureWrite : BOOL
VAR_INPUT
	input : CellDataBlock;
	mode : eModes;
END_VAR
VAR
	temp : ParameterSet; 
END_VAR
VAR CONSTANT
	indexEnablePosLimit : INT := 0;
	indexEnableNegLimit : INT := 0;
END_VAR
//command block write-in
CASE mode OF
	eModes.MODE_EXE_AXIS:
		//software limit
		fbWriteLimitPositive.Value := TO_REAL(input.axis.limitPlus) * 0.001;
		fbWriteLimitPositive.Execute := TRUE;
		
		fbWriteLimitNegtive.Value := TO_REAL(input.axis.limitMinus) * 0.001;
		fbWriteLimitNegtive.Execute := TRUE;
		
		fbEnableLimitPositive.Value := input.axis.boolParameter.indexEnablePosLimit;
		fbEnableLimitPositive.Execute := TRUE;
		
		fbEnableLimitNegtive.Value := input.axis.boolParameter.indexEnableNegLimit;
		fbEnableLimitNegtive.Execute := TRUE;
		
	eModes.MODE_EXE_COMMAND_BLOCK:
		temp := CellDataBlock2Parameter(input:= input);
		ptpCommands[input.command.base.subIndex+1] := temp; //write-in
		
END_CASE

ConfigureWrite := TRUE; //return
END_METHOD

METHOD Control : BOOL
VAR_INPUT
	input : CellDataBlock;
	mode : eModes;
END_VAR
VAR
	temp : ParameterSet;
END_VAR
//manual control servo on/servo alarm reset

//different route
CASE mode OF
	eModes.MODE_EXE_AXIS:
		IF input.axis.operationOperation.0 THEN
			//bit0ServoOn
			fbPower.Enable := NOT fbPower.Enable;
			fbPower.Enable_Positive := fbPower.Enable;
			fbPower.Enable_Negative := fbPower.Enable;
		ELSIF input.axis.operationOperation.15 THEN
			fbReset.Execute := TRUE;	
		END_IF
		Control := TRUE;
	eModes.MODE_EXE_COMMAND_BLOCK:
		temp := CellDataBlock2Parameter(input:= input);
		Control := ExecuteParameter(ptBlock:= ADR(temp));
END_CASE
END_METHOD

METHOD ErrorClear : BOOL
VAR_INPUT
	input : eErrorClearWays;
END_VAR
VAR
	nCounter : int :=1;
END_VAR
//automated mode,error reset
CASE input OF
	eErrorClearWays.RESET:
		fbReset.Execute := TRUE;
		//cancel all execution
		FOR nCounter:=1 TO 3 BY 1 DO
			fbMoveAbs[nCounter].Execute := FALSE;
		END_FOR
END_CASE
END_METHOD

METHOD ErrorDetect : UDINT
VAR_INPUT
END_VAR
VAR
	nCounter : int := 1;	
END_VAR
//Monitor all error including parameter error /drive error / logic dirve error
ErrorDetect := fbPower.ErrorID;
IF ErrorDetect = 0 THEN
	ErrorDetect := fbReadStatus.ErrorID;
END_IF
IF ErrorDetect = 0 THEN
	ErrorDetect := fbMoveHome.ErrorID;
END_IF
IF ErrorDetect = 0 THEN
	ErrorDetect := fbStop.ErrorID;
END_IF
IF ErrorDetect = 0 THEN
	ErrorDetect := fbSetPosition.ErrorID;
END_IF
//monitor all
FOR nCounter:=1 TO 3 BY 1 DO
	IF ErrorDetect = 0 THEN
		ErrorDetect := fbMoveAbs[nCounter].ErrorID;
	END_IF
END_FOR
END_METHOD

METHOD ExecuteParameter : BOOL
VAR_INPUT
	ptBlock : POINTER TO ParameterSet;
	//execute : BOOL; //used to do mutex
END_VAR
//
ExecuteParameter:=ExecuteParameterBuffer(ptBlock:= ptBlock, bufferIndex:= 1);
END_METHOD

METHOD ExecuteParameterBuffer : BOOL
VAR_INPUT
	ptBlock : POINTER TO ParameterSet;
	//execute : BOOL; //used to do mutex
	bufferIndex: INT :=1;
END_VAR
VAR
	//MC block routing
	ptMcExecute : POINTER TO BOOL;
	ptMcDone : POINTER TO BOOL;
	ptMcBusy : POINTER TO BOOL;
	ptMcError : POINTER TO BOOL;
	ptMcCommandAbort : POINTER TO BOOL;

END_VAR
//1. Do parameter translating
//2. Do command routing
//3. Control execute flow

//command routing
CASE ptBlock^.command OF
eCommandTypes.POSITION:	
	//Position command
	ptMcExecute:=ADR(fbMoveAbs[bufferIndex].Execute);
	ptMcDone:=ADR(fbMoveAbs[bufferIndex].Done);
	ptMcBusy:=ADR(fbMoveAbs[bufferIndex].Busy);
	ptMcError:=ADR(fbMoveAbs[bufferIndex].Error);
	ptMcCommandAbort := ADR(fbMoveAbs[bufferIndex].CommandAborted);
	//set once
	IF NOT fbMoveAbs[bufferIndex].Busy AND NOT ptMcExecute^ THEN
		//parameter writing
		fbMoveAbs[bufferIndex].Velocity := ptBlock^.parameter.position.Velocity;
		fbMoveAbs[bufferIndex].Acceleration:= ptBlock^.parameter.position.Acceleration;
		fbMoveAbs[bufferIndex].Deceleration:= ptBlock^.parameter.position.Deceleration;
		
		CASE ptBlock^.parameter.position.PositionType OF
			ePositionType.POSITION_ABS:
				fbMoveAbs[bufferIndex].Position := ptBlock^.parameter.position.Position;
			ePositionType.POSITION_REL:
				fbMoveAbs[bufferIndex].Position := PositionCommand + ptBlock^.parameter.position.Position; 
		END_CASE
		
	END_IF
	
	IF bufferIndex>=2 THEN
		fbMoveAbs[bufferIndex].BufferMode := MC_BlendingPrevious;
	END_IF
//torque limit
;
eCommandTypes.ZRET:
	//Home command
	ptMcExecute:=ADR(fbMoveHome.Execute);
	ptMcDone:=ADR(fbMoveHome.Done);
	ptMcBusy:=ADR(fbMoveHome.Busy);
	ptMcError:=ADR(fbMoveHome.Error);
	ptMcCommandAbort := ADR(fbMoveHome.CommandAborted);
	
	IF NOT fbMoveHome.Busy THEN
		//parameter writing
		fbMoveHome.Position := ptBlock^.parameter.home.Position;
		fbMoveHome.HomingMode := ptBlock^.parameter.home.Mode;
	END_IF
;
eCommandTypes.SET_POSITION:
	ptMcExecute:=ADR(fbSetPosition.Execute);
	ptMcDone:=ADR(fbSetPosition.Done);
	ptMcBusy:=ADR(fbSetPosition.Busy);
	ptMcError:=ADR(fbSetPosition.Error);
	ptMcCommandAbort := ADR(fbSetPosition.Done);// fake
	
	IF NOT fbSetPosition.Busy THEN
		//parameter writing
		fbSetPosition.Position := ptBlock^.parameter.position.Position;
	END_IF
	
ELSE
	return;
END_CASE

//auto stop execute when error , would do raising edge again when error eliminated
ptMcExecute^ :=  NOT ptMcDone^ ;

//power on if going to execute
IF ptMcExecute^ AND fbPower.Enable=FALSE THEN
	fbPower.Enable := TRUE;
	fbPower.Enable_Positive := TRUE;
	fbPower.Enable_Negative := TRUE;
END_IF

//done := ptMcDone^;
ExecuteParameterBuffer:=ptMcDone^; //return value
END_METHOD

METHOD ExecuteParameterBufferIndex : BOOL
VAR_INPUT
	indexCommand : INT ;
	indexBuffer : INT;
END_VAR
//wrapper function
ExecuteParameterBufferIndex := ExecuteParameterBuffer(ptBlock:= ADR(ptpCommands[indexCommand]), bufferIndex:= indexBuffer);
END_METHOD

METHOD ExecuteParameterIndex : BOOL
VAR_INPUT
	indexCommand : int;
END_VAR
//wrpper function 
ExecuteParameterIndex:=ExecuteParameter(ptBlock:= adr(ptpCommands[indexCommand]));
END_METHOD

METHOD FB_init : BOOL
VAR_INPUT
	bInitRetains : BOOL; // if TRUE, the retain variables are initialized (warm start / cold start)
	bInCopyCode : BOOL;  // if TRUE, the instance afterwards gets moved into the copy code (online change)
END_VAR
VAR
	nCounter : int ;
END_VAR
END_METHOD

METHOD Monitor : CellDataBlock
VAR_INPUT
END_VAR
Monitor.axis.operationMonitor.0 := fbPower.Enable;
Monitor.axis.operationMonitor.15 := fbReset.Execute;

Monitor.axis.runStatus.1 := fbReadStatus.StandStill;
Monitor.axis.runStatus.3 := ErrorDetect()=0;

//Monitor.axis.warning := fbReadStatus.ErrorID;
Monitor.axis.warning := ErrorDetect();

Monitor.axis.posCommand := TO_DINT(fbReadCommandPosition.Value * 1000);
Monitor.axis.posFeedback := TO_DINT(fbReadActualPosition.Position * 1000);
Monitor.axis.speedFeedback := TO_DINT(fbReadActualVelocity.Value * 1000);
Monitor.axis.torqueFeedback := TO_DINT(fbReadControlOutput.Value * 100);
END_METHOD

PROPERTY PositionCommand : LREAL
GET
fbReadCommandPosition.Enable := TRUE;
//fbReadCommandPosition(
//	Axis:= Axis, 
//	Enable:= , 
//	ParameterNumber:= CommandedPosition, 
//	ReadMode:= READMODE_ONCE, 
//	Valid=> , 
//	Busy=> , 
//	Error=> , 
//	ErrorID=> , 
//	Value=> PositionCommand);
PositionCommand := fbReadCommandPosition.Value;
END_GET
SET
END_SET
END_PROPERTY

METHOD Stop : BOOL
VAR_INPUT
END_VAR
VAR
	nCounter : INT;
END_VAR
//stop all function blocks
FOR nCounter:=1 TO 3 BY 1 DO
	fbMoveAbs[nCounter].Execute := FALSE;
END_FOR
fbMoveHome.Execute := FALSE;
fbStop.Execute := true;
END_METHOD

METHOD TypeCode : eCategrories
VAR_INPUT
END_VAR
TypeCode := eCategrories.SELECTION_AXIS;
END_METHOD

END_FUNCTION_BLOCK

// ---- POUs/Helper/Parameter2CellDataBlock.TcPOU
FUNCTION Parameter2CellDataBlock : CellDataBlock
VAR_INPUT
	input : ParameterSet;
END_VAR
VAR
END_VAR

//set command type
Parameter2CellDataBlock.command.base.commandType := input.command;

CASE input.command OF
	eCommandTypes.POSITION:
		//details setup
		IF input.parameter.position.PositionType = ePositionType.POSITION_ABS THEN
			//abs
			Parameter2CellDataBlock.command.position.controlWord.0 := 1;
		ELSE
			//rel
			Parameter2CellDataBlock.command.position.controlWord.0 := 0;
		END_IF
		IF input.parameter.position.Velocity <> 0 THEN
			Parameter2CellDataBlock.command.base.speed := TO_DWORD(input.parameter.position.Velocity / 0.001); //mm/s ->  0.001mm/s 
		END_IF
		IF input.parameter.position.Acceleration <> 0 THEN
			Parameter2CellDataBlock.command.position.accTime := TO_DWORD(( input.parameter.position.Velocity / input.parameter.position.Acceleration ) * 1000);
		END_IF
		IF input.parameter.position.Deceleration <> 0 THEN
			Parameter2CellDataBlock.command.position.decTime := TO_DWORD(( input.parameter.position.Velocity / input.parameter.position.Deceleration ) * 1000);
		END_IF
		Parameter2CellDataBlock.command.position.coordinate := TO_DWORD(input.parameter.position.Position * 1000);
	
	eCommandTypes.ZRET:
		//TODO
END_CASE

END_FUNCTION

// ---- POUs/Helper/CellDataBlock2Parameter.TcPOU
FUNCTION CellDataBlock2Parameter : ParameterSet
VAR_INPUT
	input : CellDataBlock;
END_VAR
VAR
END_VAR

//set command type
CellDataBlock2Parameter.command := input.command.base.commandType;

CASE CellDataBlock2Parameter.command OF
	eCommandTypes.POSITION:
		//details setup
		IF input.command.position.controlWord.0 THEN
			//abs
			CellDataBlock2Parameter.parameter.position.PositionType := ePositionType.POSITION_ABS;
		ELSE
			//rel
			CellDataBlock2Parameter.parameter.position.PositionType := ePositionType.POSITION_REL;	
		END_IF
		CellDataBlock2Parameter.parameter.position.Velocity := TO_LREAL(input.command.base.speed) * 0.001; //0.001mm/s -> mm/s
		IF input.command.base.accTime <> 0 THEN
			CellDataBlock2Parameter.parameter.position.Acceleration := CellDataBlock2Parameter.parameter.position.Velocity/(TO_LREAL(input.command.base.accTime) * 0.001); // ms -> mm/s2
		END_IF
		IF input.command.base.decTime <> 0 THEN
			CellDataBlock2Parameter.parameter.position.Deceleration := CellDataBlock2Parameter.parameter.position.Velocity/(TO_LREAL(input.command.base.decTime) * 0.001);
		END_IF
		CellDataBlock2Parameter.parameter.position.Position := TO_LREAL(input.command.position.coordinate) * 0.001;
	
	eCommandTypes.ZRET:
		//TODO
END_CASE

END_FUNCTION

// ---- POUs/Foundation/RunUnitGeneric.TcPOU
FUNCTION_BLOCK RunUnitGeneric Extends CommonBase
VAR_INPUT
	bEnStep : BOOL;
	bTrigStep : BOOL;
	bPause : BOOL;
	bIsBypassed : BOOL;
	bWorkingOverride : BOOL;
	bMaterialOverride : BOOL;
	
	slaveWorkingSignal : ARRAY[1..32] OF BOOL; // collect slave working signal , possible to access externally?
	
	//-------------
	//	Purge Chain
	//-------------
	isPurged : BOOL; //this station already in the purged state , would keep bypass working signals
	previousNode : POINTER TO RunUnitGeneric; // used to check previous node whether purged
END_VAR
VAR_OUTPUT
	 //possible TO output on HMI
	State AT%Q* : INT := 0;
	NextState AT%Q* : INT := 0;
	AlarmCode AT%Q* : UDINT := 0;
	WarningCode AT%Q* : UDINT := 0;
END_VAR
VAR	
	Parent : POINTER TO RunUnitGeneric;
	
	SlotBase : POINTER TO RunMaterial;
	SlotCount : INT ;
	SlotLast : POINTER TO RunMaterial;
	
	bLastParentStatus : BIT; // memorize last parent status	
	bSerialTransition : BIT;
	transitionByte : BYTE;
	
	isTransit : BOOL ;
	
	workingTimerCache : TIME;
	workingTimer : TON;
	
	outputState : INT;
	
	//do not stop in atomic operation
	atomicOperation : BOOL := FALSE;
	

END_VAR
VAR PERSISTENT
	//station specific settings area (user settings
	slaveLinkageStatus : ARRAY[1..32] OF BOOL; // configuration
	//miscsParameters : ARRAY[1..8] of int;
	
	timeoutTimer at%M* : ton; //common facility to detect time out event
END_VAR
VAR CONSTANT 
	bit0EnStep : INT := 0;
	bit1TrigStep : INT := 1;
	bit2StatePause : INT :=2;
	bit3IsBypassed : INT :=3;
	bit4WorkingOverride : INT :=4;
	bit5MaterialOverride : INT :=5;
END_VAR


//Catch parent's pause status
IF Parent<>0 AND_THEN (Parent^.bPause AND NOT bLastParentStatus) THEN
	bPause := TRUE;
END_IF

IF Parent<>0 AND_THEN (NOT Parent^.bPause AND bPause) THEN
	bPause := FALSE;
END_IF

bLastParentStatus := Parent<>0 AND_THEN Parent^.bPause;

//Serial transition
IF bSerialTransition AND (State = NextState) THEN
	NextState := State +1 ;
END_IF

//Reset transition word
IF NextState <> State THEN
	transitionByte := 0;
	bSerialTransition := FALSE;
	//AlarmCode := 0;
	
	State := NextState; //release and go
END_IF


//transit condition
isTransit := ((NOT bEnStep OR (bEnStep AND bTrigStep)) AND NOT bPause) OR atomicOperation;

IF isTransit THEN
	outputState := State; //release and go
ELSE
	outputState := eSpecialStates.FORBIDDEN;
END_IF

//Reset trigger step
bTrigStep := FALSE;

//Timer
workingTimer(IN:=,PT:=TO_TIME(4294967295),Q=>,ET=>);
timeoutTimer(IN:=,PT:=,Q=>,ET=>);
//-------------------
//purge status reset
//-------------------
IF isPurged AND (previousNode<>0 AND_THEN NOT previousNode^.isPurged) THEN
	isPurged := FALSE;
END_IF

METHOD ConfigureRead : CellDataBlock
VAR_INPUT
	input : CellDataBlock; //would offer sub-index ...etc
	mode : eModes;
END_VAR
END_METHOD

METHOD ConfigureWrite : BOOL
VAR_INPUT
	input : CellDataBlock;
	mode : eModes;
END_VAR
//Implemented by concre derived class
ConfigureWrite := true;
END_METHOD

METHOD Control : BOOL
VAR_INPUT
	input : CellDataBlock;
	mode : eModes; //commit mode
END_VAR
bEnStep := input.unit.base.controlWord.bit0EnStep;
bTrigStep := input.unit.base.controlWord.bit1TrigStep;
bPause := input.unit.base.controlWord.bit2StatePause;
bIsBypassed := input.unit.base.controlWord.bit3IsBypassed;
bWorkingOverride := input.unit.base.controlWord.bit4WorkingOverride;
bMaterialOverride := input.unit.base.controlWord.bit5MaterialOverride;
Control:=true;
END_METHOD

METHOD ErrorClear : BOOL
VAR_INPUT
	input : eErrorClearWays;
END_VAR
AlarmCode := 0; //code reset to 0
timeoutTimer.IN := false; //reset
END_METHOD

METHOD ErrorDetect : UDINT
VAR_INPUT
END_VAR
ErrorDetect := AlarmCode;
END_METHOD

METHOD FB_init : BOOL
VAR_INPUT
	bInitRetains : BOOL; // if TRUE, the retain variables are initialized (warm start / cold start)
	bInCopyCode : BOOL;  // if TRUE, the instance afterwards gets moved into the copy code (online change)
	
	argParent : POINTER TO RunUnitGeneric;
	argSlotBase : POINTER TO RunMaterial;
	argSlotLast : POINTER TO RunMaterial;
END_VAR
//initialize 
Parent := argParent;
SlotBase := argSlotBase;
SlotLast := argSlotLast;
//
IF bInitRetains THEN
	NextState := eSpecialStates.INITIAL_BEGIN;
END_IF
END_METHOD

METHOD Initialize : BOOL
VAR_INPUT
END_VAR
VAR
	nCounter : int;
END_VAR
//once initializing method call , redirect current state to initalizing region
IF (TO_UINT(State) AND TO_UINT(eSpecialStates.INITIAL_REGION)) <> 16#0100 THEN
	NextState := eSpecialStates.INITIAL_BEGIN; //not in intializing region , change
END_IF

Initialize := (State = eSpecialStates.INITIAL_END);

IF Initialize THEN
	//clear all remained signal
	FOR nCounter:=1 TO 32 BY 1 DO
		slaveWorkingSignal[nCounter] := FALSE;
	END_FOR
	//clear all internal status
	bEnStep := FALSE;
	bTrigStep := FALSE;
	bIsBypassed := FALSE;
	bWorkingOverride := FALSE;
	bMaterialOverride := FALSE;	
END_IF
END_METHOD

METHOD Monitor : CellDataBlock
VAR_INPUT
END_VAR
Monitor.unit.base.controlWord.bit0EnStep := bEnStep;
Monitor.unit.base.controlWord.bit1TrigStep := bTrigStep;
Monitor.unit.base.controlWord.bit2StatePause := bPause;
Monitor.unit.base.controlWord.bit3IsBypassed := bIsBypassed;
Monitor.unit.base.controlWord.bit4WorkingOverride := bWorkingOverride;
Monitor.unit.base.controlWord.bit5MaterialOverride := bMaterialOverride;
//Transition status
Monitor.unit.base.transitionByte := transitionByte;
//
Monitor.unit.base.alarmCode := TO_WORD(AlarmCode);
Monitor.unit.base.state := TO_WORD(State);
Monitor.unit.base.nextState := TO_WORD(NextState);
//
IF workingTimer.IN THEN
	//timer is running , reflect real value
	Monitor.unit.base.workingTimerCache := TO_DWORD(workingTimer.ET);
ELSE
	//timer is stopped , reflect cached value
	Monitor.unit.base.workingTimerCache := TO_DWORD(workingTimerCache);
END_IF
END_METHOD

METHOD TypeCode : eCategrories
VAR_INPUT
END_VAR
TypeCode := eCategrories.SELECTION_UNIT;
END_METHOD

END_FUNCTION_BLOCK

// ---- POUs/Foundation/RunMaterial.TcPOU
FUNCTION_BLOCK RunMaterial
VAR_INPUT
END_VAR
VAR_OUTPUT
END_VAR
VAR
	header AT%M* : MaterialHeader;//0-19
	block AT%M* : MaterialBlock; //20-83 (64Words
END_VAR
VAR PERSISTENT
	isNotLinked : bool; //if not linked , do not handshaking
END_VAR

PROPERTY Act : bool
GET
Act := header.wordOut.1;
END_GET
SET
IF isNotLinked THEN
	return;
END_IF

header.wordOut.1 := Act;
END_SET
END_PROPERTY

PROPERTY Data : MaterialBlock
GET
Data := block;
END_GET
SET
block := Data;
END_SET
END_PROPERTY

PROPERTY Id : DWORD
GET
Id := header.id;
END_GET
SET
header.id := Id;
END_SET
END_PROPERTY

PROPERTY Valid : bool
GET
Valid := header.wordOut.2;
END_GET
SET
header.wordOut.2 := Valid;
END_SET
END_PROPERTY

END_FUNCTION_BLOCK

// ---- DUTs/Internal/ParametersHome.TcPOU
TYPE ParametersHome :
STRUCT
	Position : LREAL := 10; // in mm
	Dummy1 : LREAL := 0;
	Dummy2 : LREAL := 0;
	Dummy3 : LREAL := 0;
	Mode : MC_HomingMode := MC_DefaultHoming;
END_STRUCT
END_TYPE

// ---- POUs/CheckBounds.TcPOU
// Implicitly generated code : DO NOT EDIT
FUNCTION CheckBounds : DINT
VAR_INPUT
	index, lower, upper: DINT;
END_VAR

// Implicitly generated code : Only an Implementation suggestion
{noflow}
IF  index < lower THEN
	CheckBounds := lower;
ELSIF  index > upper THEN
	CheckBounds := upper;
ELSE  
	CheckBounds := index;
END_IF
{flow}

END_FUNCTION

// ---- POUs/CheckPointer.TcPOU
// Implicitly generated code : DO NOT EDIT
FUNCTION CheckPointer : POINTER TO BYTE
VAR_INPUT 
	ptToTest : POINTER TO BYTE; // Destination address of the pointer
	iSize : DINT;		        // Size of the type the pointer points to. (e.g: 20 for POINTER TO ARRAY [0..9] OF INT) 
	iGran : DINT;		        // Granularity of the pointer access. This is the size of the biggest non-structured data type in the type the pointer points to. (e.g: 2 for POINTER TO ARRAY [0..9] OF INT)
	bWrite: BOOL;		        // Indicates read or write Access. TRUE = write access.
END_VAR

// No standard way of implementation. Fill your own code here
CheckPointer := ptToTest;
{flow}

END_FUNCTION

// ---- POUs/Foundation/InterfaceControlV2.TcPOU
FUNCTION_BLOCK InterfaceControlV2
VAR_INPUT
	pbStart : BOOL; //start
	pbStop : BOOL;	//stop
	pbErrorReset : BOOL; //error reset
	
	commStart AT%M* : BOOL;
	commStop AT%M* : BOOL;
	commErrorLocalAck AT%M* : BOOL; //by HMI
	commErrorIgnore AT%M* : BOOL; // by Push-button
	commErrorRemoteAck at%M* : bool;
	commInit AT%M* : BOOL;
	commPurge AT%M* : BOOL; // memorized
END_VAR
VAR_OUTPUT
	
	requestPause : BOOL;
	requestResume: BOOL;
	
	requestInit : BOOL;
	requestErrorClear : eErrorClearWays;
	
		
END_VAR

requestPause := commStop OR pbStop;
requestResume := commStart OR pbStart;

commErrorRemoteAck := pbErrorReset;

IF commErrorLocalAck OR commErrorRemoteAck THEN
	requestErrorClear := eErrorClearWays.RESET;
ELSIF commErrorIgnore THEN
	requestErrorClear := eErrorClearWays.IGNORE;
ELSE 
	//default
	requestErrorClear := eErrorClearWays.NO_ACTION;	
END_IF

//Initialization
requestInit := commInit;
//one-shot control clear 
commStart := FALSE;
commStop := FALSE;
commErrorLocalAck := FALSE;
commErrorIgnore:= FALSE;
//commInit:= FALSE;

END_FUNCTION_BLOCK

// ---- POUs/Foundation/InterfaceManualV2.TcPOU
FUNCTION_BLOCK InterfaceManualV2
VAR_INPUT
	isPaused : BOOL;
	comm : POINTER TO contextManual;
END_VAR
VAR_OUTPUT
	isManualEngaged : BOOL;
	isSemiAutoEngaged : bool;
END_VAR
VAR	
	monitorDevice : POINTER TO CommonBase;
	controlDevice : POINTER TO CommonBase;
	state : INT := 0;
	
	//need to explicit call write persistance data , to store into non-violate memory
	writePersistance : WritePersistentData;
	
	elapsed : TON ;
	m_elapsed :TIME;
	
END_VAR
VAR CONSTANT
	bEngagedHMI : INT := 0;
	bRun : INT :=1;
	bEngagedPLC : INT :=0;
	bDone : INT :=1;
END_VAR

//Write-in non-violate memory
writePersistance(
		NETID:= , 
		PORT:= 851, 
		START:= isPaused , 
		TMOUT:= , 
		BUSY=> , 
		ERR=> , 
		ERRID=> );
//---------------------------
// MONITOR
//---------------------------
IF comm^.monitorIndex >0 THEN
	CASE TO_DWORD(comm^.monitorType) OF
	eCategrories.SELECTION_AXIS:
		monitorDevice := ADR(gvl.axisControls[comm^.monitorIndex]); // index start from 1
	eCategrories.SELECTION_CYLINDER:
		monitorDevice := ADR(gvl.cylinderControls[comm^.monitorIndex]);
	eCategrories.SELECTION_VACUUM:
		monitorDevice := ADR(gvl.vacuumControls[comm^.monitorIndex]); //new type 20200228
	eCategrories.SELECTION_SIGNAL:
		monitorDevice := ADR(gvl.signalControls[comm^.monitorIndex]);
	eCategrories.SELECTION_UNIT:
		monitorDevice := ADR(gvl.units[comm^.monitorIndex]^);
	END_CASE
	comm^.monitorBlock := monitorDevice^.Monitor();
END_IF


//------------------------------
//	Control
//------------------------------
comm^.wordOut.bEngagedPLC := isPaused; //always engaged , wait
isManualEngaged:= comm^.wordIn.bEngagedHMI AND isPaused;
IF NOT  isManualEngaged THEN
	RETURN; // no longer execute further section
END_IF
isSemiAutoEngaged := isManualEngaged AND comm^.monitorType=eCategrories.SELECTION_UNIT;
//control
IF comm^.commitIndex>0 THEN
	CASE comm^.commitSelection OF
		eCategrories.SELECTION_AXIS:
			controlDevice :=  ADR(gvl.axisControls[comm^.commitIndex]);
		eCategrories.SELECTION_CYLINDER:
			controlDevice := ADR(gvl.cylinderControls[comm^.commitIndex]);
		eCategrories.SELECTION_VACUUM:
			controlDevice := ADR(gvl.vacuumControls[comm^.commitIndex]); //new type 20200228
		eCategrories.SELECTION_UNIT:
			 
			CASE comm^.commitMode OF
				eModes.MODE_DOWNLOAD_DATA_BLOCK,eModes.MODE_UPLOAD_DATA_BLOCK:
					//configuration
					controlDevice := ADR(gvl.units[comm^.commitBlock.unit.config.unitId]^);
				ELSE
					controlDevice := ADR(gvl.units[comm^.commitIndex]^);
			END_CASE
		eCategrories.SELECTION_COMMAND_BLOCK:
			//axis should be pre-selected
			controlDevice := ADR(gvl.axisControls[comm^.commitBlock.command.base.axisId]);
		eCategrories.SELECTION_SIGNAL:
			controlDevice := ADR(gvl.signalControls[comm^.commitIndex]);
	END_CASE
END_IF

CASE state OF
	0:
		IF comm^.wordIn.bEngagedHMI AND comm^.wordIn.bRun THEN
			//ENGAGED_HMI and RUN
			elapsed.IN := TRUE;		
			state := 1;
		END_IF
	1:
		IF controlDevice <>0 THEN
			CASE comm^.commitMode OF
				//Manual execution
				eModes.MODE_EXE_AXIS,eModes.MODE_EXE_COMMAND_BLOCK,eModes.MODE_EXE_CYLINDER,eModes.MODE_EXE_UNIT,eModes.MODE_EXE_VACUUM:
					comm^.wordOut.bDone := controlDevice^.Control(comm^.commitBlock,comm^.commitMode); //return whether done
				eModes.MODE_UPLOAD_DATA_BLOCK:
					comm^.commitBlock := controlDevice^.ConfigureRead(comm^.commitBlock,TO_WORD(comm^.commitSelection));
					comm^.wordOut.bDone := TRUE; //done on
				eModes.MODE_DOWNLOAD_DATA_BLOCK:
					controlDevice^.ConfigureWrite(comm^.commitBlock,TO_WORD(comm^.commitSelection));
					writePersistance.START := TRUE;
					comm^.wordOut.bDone := TRUE ;//done
				ELSE
					comm^.wordOut.bDone := TRUE ;//done
			END_CASE
		ELSE
			//null device somehow
			comm^.wordOut.bDone := TRUE;
		END_IF
		
		//interrupt operation
		IF NOT comm^.wordIn.bEngagedHMI THEN
			controlDevice^.Stop();
			comm^.wordOut.bDone := TRUE;
		END_IF
		IF comm^.wordOut.bDone THEN
			//DONE true or ENGAGED_HMI off
			m_elapsed := elapsed.ET;
			elapsed.IN := FALSE;
			state :=2;
		END_IF		
	2:
		IF NOT comm^.wordIn.bRun THEN
			comm^.wordOut.bDone := FALSE;
			state := 0;
		ELSE
			//wait RUN off
		END_IF
END_CASE

elapsed(IN:= , PT:= , Q=> , ET=> );

END_FUNCTION_BLOCK

// ---- POUs/Foundation/ProgrammedOutput.TcPOU
FUNCTION_BLOCK ProgrammedOutput
VAR_INPUT
	
	
END_VAR
VAR_OUTPUT
END_VAR
VAR
	output AT%Q* : BOOL;
	isActivated : BOOL;
	
	duty : INT;
	
	dutyCounter : INT;	
	cycleCounter : INT;
END_VAR
VAR PERSISTENT
	//output duty cycle setting
	dutiesInPercentage : ARRAY[0..3] OF INT; //multiple setting
	cycleGoal : INT;
	baseTimer : TON;
END_VAR

IF baseTimer.Q AND isActivated THEN
	dutyCounter := dutyCounter+1;
END_IF

//output when in on duty cyle
output := isActivated AND (dutyCounter < duty) AND (cycleCounter<=cycleGoal);

IF dutyCounter = duty THEN
	cycleCounter := cycleCounter +1;
END_IF

//rewind
IF dutyCounter >= 100 OR NOT isActivated THEN
	dutyCounter := 0;//reset
END_IF
IF cycleCounter >= cycleGoal OR NOT isActivated THEN
	cycleCounter := 0;//reset
END_IF

baseTimer(IN:= NOT baseTimer.Q, PT:= , Q=> , ET=> );

METHOD Activate : BOOL
VAR_INPUT
	set : int; // parameter set
END_VAR
duty := dutiesInPercentage[set];
isActivated := true;
END_METHOD

ACTION Deactivate:
isActivated := false;
END_ACTION

METHOD FB_init : BOOL
VAR_INPUT
	bInitRetains : BOOL; // if TRUE, the retain variables are initialized (warm start / cold start)
	bInCopyCode : BOOL;  // if TRUE, the instance afterwards gets moved into the copy code (online change)
END_VAR
IF bInitRetains THEN
	dutiesInPercentage[0] := 100;//always on
	dutiesInPercentage[1] := 75;//blink on
	dutiesInPercentage[2] := 50;//blink on
	dutiesInPercentage[3] := 25;//blink on
END_IF

baseTimer.PT := T#100MS; //default base
END_METHOD

END_FUNCTION_BLOCK

// ---- POUs/Foundation/RunGroupNode.TcPOU
FUNCTION_BLOCK RunGroupNode EXTENDS RunUnitGeneric
VAR_INPUT
	members : ARRAY[0..7] OF POINTER TO RunUnitGeneric;
END_VAR
VAR
	nCounter : DINT;
END_VAR

SUPER^();

CASE outputState OF 
	//------------Initialize
//	eSpecialStates.INITIAL_STATE_7:
//		// group node start initializing
//		bSerialTransition := TRUE;
		
//		//scan if all initialized
//		FOR nCounter := 0 TO 7 DO
//			IF members[nCounter] <> 0 THEN
//				bSerialTransition := bSerialTransition AND members[nCounter]^.Initialize();
//			END_IF		
//		END_FOR
		
//		// wait upper to inform starting
//		IF bSerialTransition THEN
//			NextState:=eSpecialStates.INITIAL_END;
//		END_IF

	eSpecialStates.GENERIC_GROUP_START:
		//then wait command to trigger all station into working state
		FOR nCounter := 0 TO 7 DO
			IF members[nCounter] <> 0 THEN
				members[nCounter]^.NextState := eSpecialStates.GENERIC_GROUP_START;
			END_IF
		END_FOR
		bSerialTransition := TRUE; //group idle
END_CASE

METHOD FB_init : BOOL
VAR_INPUT
	bInitRetains : BOOL; // if TRUE, the retain variables are initialized (warm start / cold start)
	bInCopyCode : BOOL;  // if TRUE, the instance afterwards gets moved into the copy code (online change)
	
	argParent : POINTER TO RunUnitGeneric;
	argSlotBase : POINTER TO RunMaterial;
	argSlotLast : POINTER TO RunMaterial;
END_VAR
//initialize 
Parent := argParent;
SlotBase := argSlotBase;
SlotLast := argSlotLast;
//
IF bInitRetains THEN
	NextState := eSpecialStates.INITIAL_BEGIN;
END_IF
END_METHOD

METHOD Initialize : BOOL
VAR_INPUT
END_VAR
VAR
	nCounter : int;
END_VAR
//once initializing method call , redirect current state to initalizing region
IF (TO_UINT(State) AND TO_UINT(eSpecialStates.INITIAL_REGION)) =0 THEN
	NextState := eSpecialStates.INITIAL_BEGIN; //not in intializing region , change
END_IF

Initialize := (State = eSpecialStates.INITIAL_END);

IF Initialize THEN
	//clear all remained signal
	FOR nCounter:=1 TO 32 BY 1 DO
		slaveWorkingSignal[nCounter] := FALSE;
	END_FOR
	//clear all internal status
	bEnStep := FALSE;
	bTrigStep := FALSE;
	bIsBypassed := FALSE;
	bWorkingOverride := FALSE;
	bMaterialOverride := FALSE;	
END_IF
END_METHOD

END_FUNCTION_BLOCK

// ---- POUs/Foundation/RunSafetyFacilityProcessor.TcPOU
FUNCTION_BLOCK RunSafetyFacilityProcessor
VAR_INPUT
	
	isPaused : BOOL; // whether auto-mode controller stopped
	
	pbReleaseSafeGuard : BOOL;
	pbEngagedSafeGuard : BOOL;
END_VAR
VAR_OUTPUT
	outPause : BOOL; //require auto-mode controller to stop
	outEmergency : BOOL; // require auto-mode controller to initialize
	outSafeGuard : BOOL; //light : safegurad  not working
	outAirAbnormal : bool; //light : air abnormal
END_VAR
VAR
	safeAck AT%Q* : BIT;
	safeRun AT%Q* : BIT;
	safeComErr AT%I* : BIT; // should trigger pause
	
	//direct status
	door1 AT%I* : BIT;
	door2 AT%I* : BIT;
	door3 AT%I* : BIT;
	door4 AT%I* : BIT;
	
	eStop1 AT%I* : BIT;
	eStop2 AT%I* : BIT;
	
	servoSto AT%I* : BIT;
	lightScreen AT%I* : BIT;
	
	//indirect status
	airChoke AT%I* : BIT;  // soft-stop valve whether activated
	safeGuardSatus AT%I* : BIT;   // should trigger pause
	eStop AT%I* : BIT;	   // should trigger initialization
	  
	//bypass
	airOff AT%Q* : BIT;
	eStopBypass AT%Q* : BIT;
	safeGuardBypass AT%Q* : BIT;
	
	//door solenoid release request
	requestSafeGuardRelease AT%I* : BOOL; //linked to HMI
	safeGuardRelease AT%Q* : BIT; //should trigger pause before, process then activate
	
	//Air valve status
	airValue1Status AT%I* : BIT;
	airValue2Status AT%I* : BIT;
	
	//mega Bypass
	outPauseBypass AT%Q* : BOOL;
	outEmergencyBypass AT%Q*: BOOL;
END_VAR

//----------------------
//	Auto resume TwinSAFE
//-----------------------
IF safeAck AND NOT safeComErr THEN
	safeAck := FALSE;
	safeRun := TRUE;
ELSIF NOT safeAck AND safeComErr THEN
	safeAck := TRUE;
	safeRun := FALSE;
END_IF

IF  safeGuardRelease AND pbEngagedSafeGuard THEN
	requestSafeGuardRelease := FALSE;
ELSIF NOT safeGuardRelease AND pbReleaseSafeGuard  AND NOT pbEngagedSafeGuard THEN
	requestSafeGuardRelease := TRUE;
ELSIF NOT isPaused then
	requestSafeGuardRelease := FALSE;
	//hold current status
END_IF
safeGuardRelease := requestSafeGuardRelease AND isPaused; //should pause firstly

outPause := (safeComErr  OR  NOT safeGuardSatus OR NOT eStop OR NOT airValue1Status OR NOT airValue2Status) AND NOT outPauseBypass;

outAirAbnormal := NOT airValue1Status OR NOT airValue2Status;
outEmergency := (safeComErr  OR NOT eStop) AND NOT outEmergencyBypass;
outSafeGuard := NOT safeGuardSatus;

END_FUNCTION_BLOCK

// ---- POUs/Foundation/RunUnitControllerV2.TcPOU
FUNCTION_BLOCK RunUnitControllerV2 EXTENDS RunGroupNode
VAR_INPUT
	isEmergency : BOOL; //would trigger initialize , raise alarm
	isSafetyFault : BOOL;
	isAirIncorrect : BOOL;
	
	isManual : BOOL;
	
	requestInit : bool;
	requestErrorClear AT%M* : eErrorClearWays := eErrorClearWays.NO_ACTION;
	
	marshal : POINTER TO RunUnitGeneric;
END_VAR
VAR_OUTPUT
	//------------------------
	//	Error handling channel
	//------------------------	
	errorType AT%Q* : eCategrories;
	errorIndex AT%Q* : DINT;
	errorCode AT%Q* : UDINT;
	
END_VAR
VAR		
	//error
	errorDevice : POINTER TO CommonBase := 0; //null reference	
	errorDelayDetect : TON;	
	
	needInit : BOOL;
END_VAR
VAR PERSISTENT
	axisUpperBound : INT;
	cylinderUpperBound : INT;
	signalUpperBound : INT;
	unitUpperBound : INT;
	slotUpperBound : int;
END_VAR
VAR CONSTANT
	ERR_EMG : DWORD :=1;
	ERR_INCORRECT_AIR : DWORD :=10;
	ERR_SAFETY : DWORD :=8501;
END_VAR

//Purpose:
// 1. As abstract machine itself , switch between modes 
// 2. bridge signals to coordinator

//Clarify : 
// 1. Manual mode : component driven only
// 2. Semi-auto (PAUSE) : sequencer were driven, but most are forbidden to execute (PAUSE state)
// 3. Auto: sequencer drive , all drive autonomous

//Difference to V1 
//1. Hierarchy initializing

//----------------------
//	Components level
//----------------------
FOR nCounter :=1 TO axisUpperBound BY 1 DO
	gvl.axisControls[nCounter]();
END_FOR
FOR nCounter :=1 TO cylinderUpperBound BY 1 DO
	gvl.pnuematicControls[nCounter]^();
END_FOR
FOR nCounter :=1 TO signalUpperBound BY 1 DO
	gvl.signalControls[nCounter]();
END_FOR
//---------------------------
//	System LEVEL
//---------------------------
IF isEmergency AND errorDelayDetect.Q   THEN
	//Emergency pressed
	//errorDevice := marshal;
	marshal^.AlarmCode := ERR_EMG;
	errorIndex := 1;
	errorDevice := marshal;
ELSIF isSafetyFault AND errorDelayDetect.Q THEN
	//Safety
	//errorDevice := marshal;
	marshal^.AlarmCode := ERR_SAFETY;
	errorIndex := 1;
	errorDevice := marshal;
ELSIF isAirIncorrect AND errorDelayDetect.Q  THEN
	//Air supply
	//errorDevice := marshal;
	marshal^.AlarmCode := ERR_INCORRECT_AIR;
	errorIndex := 1;
	errorDevice := marshal;
ELSE
	//----------------------------------------
	// 	COMPONENT LEVEL:
	//	running all devices/detect errors
	//----------------------------------------
	FOR nCounter :=1 TO axisUpperBound BY 1 DO
		//error detection
		IF errorDevice=0 AND errorDelayDetect.Q AND gvl.axisControls[nCounter].ErrorDetect() <> 0 THEN
			//error scaned
			errorIndex := nCounter;
			errorDevice := ADR(gvl.axisControls[nCounter]);
		END_IF
	END_FOR
	FOR nCounter :=1 TO cylinderUpperBound BY 1 DO
		//error detection
		IF errorDevice=0 AND errorDelayDetect.Q AND gvl.pnuematicControls[nCounter]^.ErrorDetect() <> 0 THEN
			//error scaned
			errorIndex := nCounter;
			errorDevice := gvl.pnuematicControls[nCounter];
		END_IF
	END_FOR
	FOR nCounter :=1 TO unitUpperBound BY 1 DO
		//error detection
		IF errorDevice=0 AND errorDelayDetect.Q AND gvl.units[nCounter] <> 0 AND_THEN gvl.units[nCounter]^.ErrorDetect() <> 0THEN
			//station
			errorIndex := nCounter;
			errorDevice := gvl.units[nCounter];
		END_IF
	END_FOR
END_IF


//routines
errorDelayDetect(IN:= (errorDevice = 0), PT:= T#200MS, Q=> , ET=> );	//after reset , wait 100ms to detect
IF errorDevice <>0 THEN
	//error index had been specified
	errorType := errorDevice^.TypeCode();
	errorCode := errorDevice^.ErrorDetect();
	
	//reset error handling
	IF requestErrorClear <> eErrorClearWays.NO_ACTION THEN
		errorDevice^.ErrorClear(requestErrorClear); //call error clear function
		errorDevice := 0 ;// cut link
	END_IF
	
	
ELSE
	//reset
	errorType := 0;
	errorIndex := 0;
	errorCode := 0;
END_IF
AlarmCode := SHL(TO_UDINT(errorType),24) +  TO_UDINT(SHL(errorIndex,16)) + TO_UDINT(errorCode);

//-------------------------------------------------
// START/STOP (internal pause due to process error
//-------------------------------------------------
IF errorDevice <>0  THEN
	bPause := TRUE; //forced stop
ELSE
	//leave current status
END_IF
//------------------------------------------------------------
//	IN MANUAL MODE, FORBIDEEN TO DRIVE SEQUENCES
//------------------------------------------------------------
IF NOT isManual THEN
	// sequences driven
	FOR nCounter :=1 TO unitUpperBound BY 1 DO
		IF gvl.units[nCounter] <> 0 THEN
			gvl.units[nCounter]^();
		END_IF
	END_FOR
END_IF

//-------------------
//	Check whether init condition
//, TODO or fatal situation
//-------------------
IF NOT needInit AND isEmergency THEN
	needInit := TRUE;
END_IF

SUPER^(); //state machine driven
CASE outputState OF
	eSpecialStates.MAIN_WAIT_INITIALIZING:
		bSerialTransition := requestInit AND NOT isEmergency;
		IF bSerialTransition THEN
			needInit := FALSE; //reset
		END_IF
	eSpecialStates.MAIN_INITIALIZING:
		bSerialTransition := marshal<>0 AND_THEN marshal^.Initialize();
		IF bSerialTransition THEN
			marshal^.NextState := eSpecialStates.GENERIC_GROUP_START;
		END_IF
	eSpecialStates.MAIN_INITIALIZED:
		//wait emergency situation 
		IF needInit OR requestInit THEN
			NextState := eSpecialStates.MAIN_WAIT_INITIALIZING;
		END_IF
END_CASE

METHOD FB_init : BOOL
VAR_INPUT
	bInitRetains : BOOL; // if TRUE, the retain variables are initialized (warm start / cold start)
	bInCopyCode : BOOL;  // if TRUE, the instance afterwards gets moved into the copy code (online change)
	
	argParent : POINTER TO RunUnitGeneric;
	argSlotBase : POINTER TO RunMaterial;
	argSlotLast : POINTER TO RunMaterial;
	
END_VAR
//initialize 
Parent := argParent;
SlotBase := argSlotBase;
SlotLast := argSlotLast;
//
IF bInitRetains THEN
	NextState := eSpecialStates.INITIAL_BEGIN;
	
	// Semi-statically setup running index bound
	axisUpperBound := SIZEOF(gvl.axisControls)/SIZEOF(gvl.axisControls[1]);
	cylinderUpperBound := SIZEOF(gvl.cylinderControls)/SIZEOF(gvl.cylinderControls[1]);
	signalUpperBound := SIZEOF(gvl.signalControls)/SIZEOF(gvl.signalControls[1]);
	unitUpperBound := SIZEOF(gvl.units)/SIZEOF(gvl.units[1]);
	slotUpperBound := SIZEOF(gvl.materialSlots)/SIZEOF(gvl.materialSlots[1]);
	
END_IF

state := eSpecialStates.MAIN_INITIALIZING; //as beginning
NextState:=state;
END_METHOD

END_FUNCTION_BLOCK

// ---- POUs/Foundation/RunUnitSlave.TcPOU
FUNCTION_BLOCK RunUnitSlave EXTENDS RunUnitGeneric
VAR
	workingSignal : POINTER TO BOOL;  // start working when on
END_VAR

SUPER^();

CASE outputState OF 
	eSpecialStates.SLAVE_WORK_TRIGGER:
		//working start
		IF workingSignal<>0 AND_THEN workingSignal^ THEN		
			bWorkingOverride := TRUE; // backup working override signal
		END_IF
		IF bWorkingOverride AND NOT bIsBypassed THEN
			NextState := eSpecialStates.SLAVE_ENTER_PROCEDURE; // enter working procedure
			workingSignal^ := TRUE;
			workingTimer.IN := TRUE;
			//--------------------
			//	Material override
			//--------------------
			IF SlotBase<>0 AND_THEN SlotBase^.Valid THEN
				bMaterialOverride := TRUE;
			END_IF			
		ELSIF bWorkingOverride AND bIsBypassed THEN
			NextState := eSpecialStates.SLAVE_WORK_DONE;
		ELSE
			//do nothing
		END_IF
		
	eSpecialStates.SLAVE_WORK_DONE:
		//working done
		workingSignal^ := FALSE;
		bMaterialOverride := FALSE;
		NextState := eSpecialStates.SLAVE_WORK_TRIGGER; // rewind
END_CASE

//sychoronizing
IF NOT workingSignal^ AND bWorkingOverride THEN
	bWorkingOverride := FALSE;
END_IF

//stop watch
IF workingTimer.IN AND NOT bWorkingOverride THEN
	workingTimerCache := workingTimer.ET;
	workingTimer.IN := FALSE;
END_IF

METHOD FB_init : BOOL
VAR_INPUT
	bInitRetains : BOOL; // if TRUE, the retain variables are initialized (warm start / cold start)
	bInCopyCode : BOOL;  // if TRUE, the instance afterwards gets moved into the copy code (online change)
	
	argParent : POINTER TO RunUnitGeneric;
	argSlotBase : POINTER TO RunMaterial;
	argSlotLast : POINTER TO RunMaterial;
	
	argWorkingSignal : POINTER TO BOOL;
END_VAR
//initialize 
Parent := argParent;
SlotBase := argSlotBase;
SlotLast := argSlotLast;
//
IF bInitRetains THEN
	NextState := eSpecialStates.INITIAL_BEGIN;
END_IF

workingSignal := argWorkingSignal; //link
END_METHOD

END_FUNCTION_BLOCK

// ---- POUs/Foundation/RunVacuum.TcPOU
FUNCTION_BLOCK RunVacuum EXTENDS ExecuteBase
VAR_INPUT
	isErrorDetectEnabled : BOOL;
	isActiveAutoBreakStroke : BOOL;	//TODO , start breaker stroke then stop
END_VAR
VAR_OUTPUT
	vacuumSensorValue AT %I* : UINT;
END_VAR
VAR
	COMMAND_CACHED : eCylinderCommands; //1 , HMI->PLC
	LAST_COMMAND : eCylinderCommands;   //2 , 
		
	ACT_GENERATOR AT %Q* : BOOL;
	ACT_BREAKER AT %Q* : BOOL;
		
	thresholdsMatches: ARRAY[0..3] OF BOOL; //numerical in
	thresholdMatched : BOOL;
	
	nCounter : INT := 0;
	bMatched : BOOL := false;
		
	BIT_WARNING : BOOL; //0	
	BIT_WARN_SUPPRESS : BOOL; //3 , (Control)
	BIT_DONE : BOOL; //5 (Threshold matched)
	
	isMatched : BOOL;
	isStrokeReach : BOOL;
END_VAR
VAR PERSISTENT
	thresholdCurrentSet : INT; //
	thresholdValues : ARRAY[0..3] OF UINT;
	
	TMR_WATCH_DOG : TON ; //Watch dog timer
	TMR_DELAY_TO_THRESHOLD : TON;
	TMR_DELAY_TO_OFF : TON;
END_VAR

SUPER^();

//Command received -> delay -> output , and refresh relative sensor

//------------
//
//-------------
FOR nCounter:= 0 TO 3 BY 1 DO
	thresholdsMatches[nCounter] := (vacuumSensorValue >= thresholdValues[nCounter]);
END_FOR
// scan all sensor status
thresholdMatched := thresholdsMatches[thresholdCurrentSet]; // whether match the master set
//Run timers
TMR_WATCH_DOG(IN:= , PT:= , Q=> , ET=> );
TMR_DELAY_TO_THRESHOLD(IN:= , PT:= , Q=> , ET=> );
TMR_DELAY_TO_OFF(IN:= , PT:= , Q=> , ET=> );

IF NOT TMR_DELAY_TO_THRESHOLD.IN THEN
	TMR_DELAY_TO_THRESHOLD.IN := TRUE;
END_IF

// once command changes , reset timer counter
IF COMMAND_CACHED <> LAST_COMMAND THEN
	//reset done/warn
	BIT_DONE := FALSE;
	BIT_WARNING := FALSE;
	
	//output 
	ACT_BREAKER := (COMMAND_CACHED = eCylinderCommands.COMMAND_A);
	ACT_GENERATOR := (COMMAND_CACHED = eCylinderCommands.COMMAND_B);
	
	TMR_DELAY_TO_THRESHOLD.IN := (COMMAND_CACHED=eCylinderCommands.COMMAND_B);
	TMR_DELAY_TO_OFF.IN := (COMMAND_CACHED=eCylinderCommands.COMMAND_A);
END_IF


//reset
bMatched := FALSE;
// Check if match
CASE COMMAND_CACHED OF
	eCylinderCommands.NO_COMMAND,eCylinderCommands.COMMAND_A:
		bMatched:= TRUE;
	
	eCylinderCommands.COMMAND_B:
	
		bMatched:= (thresholdMatched ) ; //AND TMR_DELAY_TO_THRESHOLD.Q;
	
		
END_CASE

//start
IF NOT bMatched AND TMR_DELAY_TO_THRESHOLD.Q THEN
	TMR_WATCH_DOG.in := TRUE;
ELSE
	TMR_WATCH_DOG.in := FALSE;
END_IF

isMatched :=  bMatched OR (NOT bMatched AND BIT_WARN_SUPPRESS );
isStrokeReach :=  (COMMAND_CACHED=eCylinderCommands.COMMAND_B AND TMR_DELAY_TO_THRESHOLD.Q) OR (COMMAND_CACHED=eCylinderCommands.COMMAND_A AND TMR_DELAY_TO_OFF.Q)  OR COMMAND_CACHED=eCylinderCommands.NO_COMMAND;
// status update
//BIT_DONE := isShutVerification OR (bMatched OR (NOT bMatched AND (BIT_WARN_SUPPRESS  ) AND TMR_WATCH_DOG.Q));
//BIT_WARNING := NOT isShutVerification AND(NOT bMatched) AND (NOT BIT_WARN_SUPPRESS) AND TMR_WATCH_DOG.Q AND TMR_DELAY_TO_THRESHOLD.Q;
BIT_DONE := isShutVerification OR isMatched AND isStrokeReach;
BIT_WARNING := NOT isShutVerification AND NOT isMatched AND TMR_WATCH_DOG.Q ;


// cache last command
LAST_COMMAND := COMMAND_CACHED;

METHOD ConfigureRead : CellDataBlock
VAR_INPUT
	input : CellDataBlock; //would offer sub-index ...etc
	mode : eModes;
END_VAR

ConfigureRead.vacuum.threshold := TO_WORD(thresholdValues[0]);
ConfigureRead.vacuum.timerSetValue := TO_WORD(TMR_DELAY_TO_THRESHOLD.PT);
END_METHOD

METHOD ConfigureWrite : BOOL
VAR_INPUT
	input : CellDataBlock;
	mode : eModes;
END_VAR

TMR_DELAY_TO_THRESHOLD.PT := TO_TIME(input.vacuum.timerSetValue);
thresholdValues[0] := input.vacuum.threshold;
END_METHOD

METHOD Control : BOOL
VAR_INPUT
	input : CellDataBlock;
	mode : eModes;
END_VAR
Execute(argCommand:= input.cylinder.command);
Control:=true;
END_METHOD

METHOD ErrorClear : BOOL
VAR_INPUT
	input : eErrorClearWays;
END_VAR
//suppress is the only way
BIT_WARN_SUPPRESS := TRUE;
END_METHOD

METHOD ErrorDetect : UDINT
VAR_INPUT
END_VAR
IF NOT isErrorDetectEnabled THEN
	ErrorDetect := 0;
ELSIF BIT_WARNING THEN
	ErrorDetect := COMMAND_CACHED; //distinguish different error 
END_IF
END_METHOD

METHOD Execute : BOOL
VAR_INPUT
	argCommand : eCylinderCommands;
END_VAR
VAR
	outDone : BOOL ;
END_VAR
// store command
COMMAND_CACHED := argCommand;

outDone := BIT_DONE AND NOT BIT_WARNING AND (COMMAND_CACHED = LAST_COMMAND);

//reset surpress
IF outDone THEN
	BIT_WARN_SUPPRESS := FALSE;
END_IF

Execute:=outDone; //return
END_METHOD

METHOD FB_init : BOOL
VAR_INPUT
	bInitRetains : BOOL; // if TRUE, the retain variables are initialized (warm start / cold start)
	bInCopyCode : BOOL;  // if TRUE, the instance afterwards gets moved into the copy code (online change)
	
	//argASensorUsed : INT := 0;
	//argBSensorUsed : INT := 0;
END_VAR
VAR
	nCounter : int;
END_VAR
//A_SENSOR_USED_COUNT := argASensorUsed;
//B_SENSOR_USED_COUNT := argBSensorUsed;

//given timer initial value
//TMR_WATCH_DOG.PT := T#200MS;
//TMR_DELAY_TO_A.PT := T#200MS;
//TMR_DELAY_TO_B.PT := T#200MS;
IF bInitRetains THEN
	TMR_WATCH_DOG.PT := T#200MS;
	TMR_DELAY_TO_THRESHOLD.PT := T#200MS;
	
	thresholdCurrentSet := 0;
	
	FOR nCounter:= 0 TO 15 BY 1 DO
		thresholdValues[nCounter] := -1; 
// default thresholds less than default read-in
// would always output MATCHED
	END_FOR
END_IF
END_METHOD

METHOD Monitor : CellDataBlock
VAR_INPUT
END_VAR
VAR CONSTANT
	bit0Warn : INT :=0;
	bit1MonGroupA : INT :=1;
	bit2MonGroupB : INT :=2;
	bit3CtlSuppress : INT :=3;
	bit4TmrOn : INT :=4;
	bit5Done : INT := 5;
	//New
	bit6TmrAOn : INT :=6;
	bit7TmrBOn : INT :=7;
END_VAR
VAR
	TMR_DELAY_TO_B: INT;
END_VAR
//TODO , reserved

Monitor.vacuum.statusWord.bit0Warn := BIT_WARNING;
//Monitor.vacuum.statusWord.bit1MonGroupA := BIT_A_MATCH;
//Monitor.vacuum.statusWord.bit2MonGroupB := BIT_B_MATCH;
Monitor.vacuum.statusWord.bit3CtlSuppress := BIT_WARN_SUPPRESS;
Monitor.vacuum.statusWord.bit4TmrOn := TMR_WATCH_DOG.Q;
Monitor.vacuum.statusWord.bit5Done := BIT_DONE;

//Monitor.vacuum.statusWord.bit6TmrAOn := TMR_DELAY_TO_A.Q;
//Monitor.vacuum.statusWord.bit7TmrBOn := TMR_DELAY_TO_B.Q;

Monitor.vacuum.lastCommand := LAST_COMMAND;
//Monitor.vacuum.
Monitor.vacuum.vacuumValue := vacuumSensorValue;
END_METHOD

METHOD TypeCode : eCategrories
VAR_INPUT
END_VAR
TypeCode := eCategrories.SELECTION_VACUUM;
END_METHOD

END_FUNCTION_BLOCK

// ---- POUs/Foundation/SemephoreV1.TcPOU
FUNCTION_BLOCK SemephoreV1
VAR_INPUT
	currentMode : eOperationModes;
	isError : BOOL;
	isInitializing : BOOL;
END_VAR
VAR_OUTPUT
END_VAR
VAR
	io : POINTER TO ioBundleControl;
	buzzerCounter : INT;
END_VAR
VAR PERSISTENT
	buzzerTimerOn : TON;
	buzzerTimerOff : TON;
	buzzerGoal : INT := 5;
	buzzerEnable : bool := false;
END_VAR

//reset all
io^.lightGreen := FALSE;
io^.lightRed := FALSE;
io^.lightYellow := FALSE;
io^.lightWhite := FALSE;
io^.towerGreen := FALSE;
io^.towerRed := FALSE;
io^.towerYellow := FALSE;
//io^.towerBuzzer := FALSE;

CASE currentMode OF
	eOperationModes.AUTO:
		io^.lightGreen := TRUE;
	eOperationModes.MANUAL,eOperationModes.SEMI_AUTO:
		io^.lightRed := TRUE;
		io^.towerYellow := TRUE;
END_CASE

io^.lightYellow := isError OR isInitializing;
io^.towerRed := isError;
io^.towerYellow := io^.towerYellow OR isInitializing;
io^.towerGreen := NOT io^.towerRed AND NOT io^.towerYellow;

//buzser (fliper
buzzerTimerOn(IN:= , PT:= , Q=>, ET=> );
buzzerTimerOff(IN:= , PT:= , Q=> , ET=> );

IF buzzerTimerOn.Q THEN
	buzzerTimerOff.IN := TRUE;
	buzzerTimerOn.IN := FALSE;
ELSIF buzzerTimerOff.Q THEN
	buzzerTimerOff.IN := FALSE;
	buzzerTimerOn.IN := TRUE;
	
	buzzerCounter := buzzerCounter +1; // a cycle complished
	
ELSIF NOT buzzerTimerOn.IN AND NOT buzzerTimerOff.IN THEN
	buzzerTimerOn.IN := TRUE;
END_IF

IF  NOT isError THEN
	buzzerCounter := 0;
END_IF
// error comes and timeron and counter not reached
io^.towerBuzzer := isError AND buzzerTimerOn.Q AND (buzzerCounter < buzzerGoal) and buzzerEnable;

METHOD FB_init : BOOL
VAR_INPUT
	bInitRetains : BOOL; // if TRUE, the retain variables are initialized (warm start / cold start)
	bInCopyCode : BOOL;  // if TRUE, the instance afterwards gets moved into the copy code (online change)
	
	argIo : pointer to ioBundleControl;
END_VAR
io := argIo;
END_METHOD

END_FUNCTION_BLOCK

// ---- POUs/Foundation/SemephoreV2.TcPOU
FUNCTION_BLOCK SemephoreV2
VAR_INPUT
	isPaused : BOOL;
	isError : BOOL;
	isWarning : BOOL;
	isInitializing : BOOL;
	
	isDoorOpen : BOOL;
	//------------------
	//	Pushbutton lighter
	//------------------
	lightRed AT%Q* : BIT; //being paused
	lightGreen AT%Q* : BIT;
	lightYellow AT%Q* : BIT;
	lightWhite AT%Q* : BIT;
END_VAR
VAR
	buzzerCounter : INT;
	
	//----------------
	//	Towers
	//----------------
	towerRed AT%Q* : BIT;
	towerGreen AT%Q* : BIT;
	towerYellow AT%Q* : BIT;
	towerBuzzer AT%Q* : BIT;
	
END_VAR
VAR PERSISTENT
	buzzerTimerOn : TON;
	buzzerTimerOff : TON;
	buzzerGoal : INT := 5;
	buzzerEnable AT%M*: BOOL := FALSE;
END_VAR

towerRed := isError;
towerYellow := isPaused OR isInitializing;
towerGreen := NOT towerRed AND NOT towerYellow;

lightGreen := NOT isPaused;
lightRed := NOT lightGreen;
lightYellow := isError;
lightWhite := isDoorOpen;

//buzser (fliper
buzzerTimerOn(IN:= , PT:= , Q=>, ET=> );
buzzerTimerOff(IN:= , PT:= , Q=> , ET=> );

IF buzzerTimerOn.Q THEN
	buzzerTimerOff.IN := TRUE;
	buzzerTimerOn.IN := FALSE;
ELSIF buzzerTimerOff.Q THEN
	buzzerTimerOff.IN := FALSE;
	buzzerTimerOn.IN := TRUE;
	
	buzzerCounter := buzzerCounter +1; // a cycle complished
	
ELSIF NOT buzzerTimerOn.IN AND NOT buzzerTimerOff.IN THEN
	buzzerTimerOn.IN := TRUE;
END_IF

IF  NOT isError THEN
	buzzerCounter := 0;
END_IF
// error comes and timeron and counter not reached
towerBuzzer := isError AND buzzerTimerOn.in AND (buzzerCounter < buzzerGoal) AND buzzerEnable;

END_FUNCTION_BLOCK

// ---- POUs/Foundation/InterfaceControlV1.TcPOU
FUNCTION_BLOCK InterfaceControlV1
VAR_INPUT
	currentMode : eOperationModes;
	pbGreen : BOOL; //start
	pbRed : BOOL;	//stop
	pbYellow: BOOL; //error reset
	//
	errorType : DWORD;
	errorIndex : DWORD;
	errorCode : LWORD;
	//
	state : WORD;
END_VAR
VAR_OUTPUT
	requestMode : eOperationModes;
	requestInit : BOOL;
	errorClear : eErrorClearWays;
	
	materialClear : BOOL;
		
END_VAR
VAR
	comm AT%MB256 : commUnitController;
	
	errorCodePointer : POINTER TO DWORD;
END_VAR
VAR CONSTANT
	bErrorReset : INT := 0;
	bPause : INT :=1;
	bInitialize : INT :=2;
	bManualMode : INT :=3;
	bErrorIgnore : INT :=4;
	bClear : INT :=5;
END_VAR

//Start/Stop/Manual

//default request mode = current mode
requestMode := currentMode;

CASE currentMode OF
	eOperationModes.AUTO:
		IF comm.control.bPause OR pbRed THEN
			requestMode := eOperationModes.SEMI_AUTO;
		END_IF
		comm.controlWord.2 := FALSE; //pause state
	eOperationModes.SEMI_AUTO:
		IF comm.control.bManualMode THEN
			//higher priority
			requestMode := eOperationModes.MANUAL;
		ELSIF comm.control.bPause OR pbGreen THEN
			requestMode := eOperationModes.AUTO;
		END_IF
		comm.controlWord.2 := TRUE; //pause state
	eOperationModes.MANUAL:
		IF not comm.control.bManualMode THEN
			requestMode := eOperationModes.SEMI_AUTO;
		END_IF
		comm.controlWord.2 := TRUE; //pause state
END_CASE
//Initialization
requestInit := comm.control.bInitialize;
//Error clear request
errorClear := eErrorClearWays.NO_ACTION;
IF comm.control.bErrorReset OR pbYellow THEN
	errorClear := eErrorClearWays.RESET;
ELSIF comm.control.bErrorIgnore THEN
	errorClear := eErrorClearWays.IGNORE;	
END_IF
//material clear
materialClear := comm.control.bClear; 
//one-shot control clear , except bManualMode
comm.control := 16#8 AND comm.control;
//error infomation
comm.errorType := errorType;
comm.errorIndex := errorIndex;
errorCodePointer := ADR(errorCode);
comm.errorCode1 := errorCodePointer[0]; //seperated
comm.errorCode2 := errorCodePointer[1]; //seperated
//
comm.state := state;

METHOD ErrorInfomation : BOOL
VAR_INPUT
	mErrorIndex : INT;
	mErrorType : eCategrories;
	mErrorCode : UDINT;
END_VAR
comm.errorIndex := TO_DWORD(mErrorIndex);
comm.errorType := mErrorType;
comm.errorCode1 := mErrorCode;
END_METHOD

METHOD MonitorData : DWORD
VAR_INPUT
	index : INT;
	value : DWORD;
END_VAR
comm.monitorDatas[index] := value;
END_METHOD

END_FUNCTION_BLOCK

// ---- POUs/Foundation/InterfaceManualV1.TcPOU
FUNCTION_BLOCK InterfaceManualV1
VAR_INPUT
	currentMode : eOperationModes;
END_VAR
VAR_OUTPUT
END_VAR
VAR

	comm AT%MB1024: commManual;
	
	monitorDevice : POINTER TO CommonBase;
	controlDevice : POINTER TO CommonBase;
	state : INT := 0;
	
	//need to explicit call write persistance data , to store into non-violate memory
	writePersistance : WritePersistentData;
	
	elapsed : TON ;
	m_elapsed :TIME;
END_VAR
VAR CONSTANT
	bEngagedHMI : INT := 0;
	bRun : INT :=1;
	bEngagedPLC : INT :=0;
	bDone : INT :=1;
END_VAR

IF writePersistance.START And not writePersistance.BUSY THEN
	writePersistance.START := false;
END_IF
//Write-in non-violate memory
writePersistance(
		NETID:= , 
		PORT:= 851, 
		START:= , 
		TMOUT:= , 
		BUSY=> , 
		ERR=> , 
		ERRID=> );

//
CASE currentMode OF
	eOperationModes.AUTO:
		comm.wordOut.bEngagedPLC := FALSE;
		RETURN;
	ELSE
		//MANUAL and SEMI-AUTO
		comm.wordOut.bEngagedPLC := TRUE;
END_CASE
//monitor
CASE TO_DWORD(comm.monitorType) OF
	eCategrories.SELECTION_AXIS:
		monitorDevice := ADR(gvl.axisControls[comm.monitorIndex+1]); // index start from 1
	eCategrories.SELECTION_CYLINDER:
		monitorDevice := ADR(gvl.cylinderControls[comm.monitorIndex+1]);
	eCategrories.SELECTION_SIGNAL:
		monitorDevice := ADR(gvl.signalControls[comm.monitorIndex+1]);
	eCategrories.SELECTION_UNIT:
		monitorDevice := ADR(gvl.units[comm.monitorIndex+1]^);
END_CASE
comm.monitorBlock := monitorDevice^.Monitor();
//control
CASE comm.commitSelection OF
	eCategrories.SELECTION_AXIS:
		controlDevice :=  ADR(gvl.axisControls[comm.commitIndex+1]);
	eCategrories.SELECTION_CYLINDER:
		controlDevice := ADR(gvl.cylinderControls[comm.commitIndex+1]);
	eCategrories.SELECTION_UNIT:
		 
		CASE comm.commitMode OF
			eModes.MODE_DOWNLOAD_DATA_BLOCK,eModes.MODE_UPLOAD_DATA_BLOCK:
				//configuration
				controlDevice := ADR(gvl.units[comm.commitBlock.unit.config.unitId+1]^);
			ELSE
				controlDevice := ADR(gvl.units[comm.commitIndex+1]^);
		END_CASE
	eCategrories.SELECTION_COMMAND_BLOCK:
		//axis should be pre-selected
		controlDevice := ADR(gvl.axisControls[comm.commitBlock.command.base.axisId+1]);
	eCategrories.SELECTION_SIGNAL:
		controlDevice := ADR(gvl.signalControls[comm.commitIndex+1]);
END_CASE
CASE state OF
	0:
		IF comm.wordIn.bEngagedHMI AND comm.wordIn.bRun THEN
			//ENGAGED_HMI and RUN
			elapsed.IN := TRUE;		
			state := 1;
		END_IF
	1:
		CASE comm.commitMode OF
				//Manual execution
				eModes.MODE_EXE_AXIS,eModes.MODE_EXE_COMMAND_BLOCK,eModes.MODE_EXE_CYLINDER,eModes.MODE_EXE_UNIT:
					comm.wordOut.bDone := controlDevice^.Control(comm.commitBlock,comm.commitMode); //return whether done
				eModes.MODE_UPLOAD_DATA_BLOCK:
					comm.commitBlock := controlDevice^.ConfigureRead(comm.commitBlock,TO_WORD(comm.commitSelection));
					comm.wordOut.bDone := TRUE; //done on
				eModes.MODE_DOWNLOAD_DATA_BLOCK:
					controlDevice^.ConfigureWrite(comm.commitBlock,TO_WORD(comm.commitSelection));
					writePersistance.START := TRUE;
					comm.wordOut.bDone := TRUE ;//done
				ELSE
					comm.wordOut.bDone := TRUE ;//done
		END_CASE
		//interrupt operation
		IF NOT comm.wordIn.bEngagedHMI THEN
			controlDevice^.Stop();
			comm.wordOut.bDone := TRUE;
		END_IF
		IF comm.wordOut.bDone THEN
			//DONE true or ENGAGED_HMI off
			m_elapsed := elapsed.ET;
			elapsed.IN := FALSE;
			state :=2;
		END_IF		
	2:
		IF NOT comm.wordIn.bRun THEN
			comm.wordOut.bDone := FALSE;
			state := 0;
		ELSE
			//wait RUN off
		END_IF
END_CASE

elapsed(IN:= , PT:= , Q=> , ET=> );

END_FUNCTION_BLOCK

// ---- POUs/Foundation/RunUnitControllerV1.TcPOU
FUNCTION_BLOCK RunUnitControllerV1 EXTENDS RunUnitGeneric
VAR_INPUT
END_VAR
VAR_OUTPUT
	currentMode : eOperationModes := eOperationModes.MANUAL; //default in semi-auto
	isInitializing : BOOL;
	isError : BOOL;
	
END_VAR
VAR		
	nCounter : INT;
	bAllInitialized : BOOL := FALSE;
	
	//user control
	requestInitialize : BOOL;
	//error
	requestErrorClear : eErrorClearWays := eErrorClearWays.NO_ACTION;
	errorDevice : POINTER TO CommonBase := 0; //null reference
	errorType : eCategrories;
	errorIndex : INT;
	errorCode : UDINT;
	errorDelayDetect : TON;	
	//HMI Control interface
	interfaceControl : POINTER TO InterfaceControlV1;
	interfaceManual : POINTER TO InterfaceManualV1;
	
	pbRed : POINTER TO RunSignal;
	pbGreen : POINTER TO RunSignal;
	pbYellow : POINTER TO RunSignal;
END_VAR
VAR PERSISTENT
	axisUpperBound : INT;
	cylinderUpperBound : INT;
	signalUpperBound : INT;
	unitUpperBound : INT;
	slotUpperBound : int;
END_VAR

//scan running all devices
FOR nCounter :=1 TO axisUpperBound BY 1 DO
	gvl.axisControls[nCounter]();
	//error detection
	IF errorDevice=0 AND errorDelayDetect.Q AND gvl.axisControls[nCounter].ErrorDetect() <> 0 THEN
		//error scaned
		interfaceControl^.errorIndex := TO_DWORD(nCounter-1);
		errorDevice := ADR(gvl.axisControls[nCounter]);
	END_IF
END_FOR
FOR nCounter :=1 TO cylinderUpperBound BY 1 DO
	gvl.cylinderControls[nCounter]();
	//error detection
	IF errorDevice=0 AND errorDelayDetect.Q AND gvl.cylinderControls[nCounter].ErrorDetect() <> 0 THEN
		//error scaned
		interfaceControl^.errorIndex := TO_DWORD(nCounter-1);
		errorDevice := ADR(gvl.cylinderControls[nCounter]);
	END_IF
END_FOR
FOR nCounter :=1 TO signalUpperBound BY 1 DO
	gvl.signalControls[nCounter]();
END_FOR
FOR nCounter :=1 TO unitUpperBound BY 1 DO
	//error detection
	IF errorDevice=0 AND errorDelayDetect.Q AND gvl.units[nCounter] <> 0 AND_THEN gvl.units[nCounter]^.ErrorDetect() <> 0THEN
		//station
		interfaceControl^.errorIndex := TO_DWORD(nCounter-1);
		errorDevice := gvl.units[nCounter];
	END_IF
END_FOR
//routines
errorDelayDetect(IN:= (errorDevice = 0), PT:= T#100MS, Q=> , ET=> );	//after reset , wait 100ms to detect
IF errorDevice <>0 THEN
	//errorIndex := nCounter-1;
	interfaceControl^.errorType := errorDevice^.TypeCode();
	interfaceControl^.errorCode := errorDevice^.ErrorDetect();
		
	ErrorHandler();// handling user-input reset/ignore
ELSE
	//reset
	interfaceControl^.errorType := 0;
	interfaceControl^.errorIndex := 0;
	interfaceControl^.errorCode := 0;
END_IF
isError := errorDevice <>0;
//reflect to interface
interfaceManual^(
	currentMode:= THIS^.currentMode); //scan-in,scan-out,manual...
//handling input request
interfaceControl^(
	currentMode:= THIS^.currentMode,
	pbGreen := pbGreen^.debouncedOn,
	pbRed := pbRed^.debouncedOn,
	pbYellow := pbYellow^.debouncedOn,
	errorClear=> THIS^.requestErrorClear);
IF interfaceControl^.requestInit THEN
	requestInitialize := TRUE; // memorize
END_IF
//mode switcher pre-check
bPause := NOT (currentMode = eOperationModes.AUTO);
IF interfaceControl^.requestMode <> currentMode THEN
	CASE interfaceControl^.requestMode OF 
		eOperationModes.MANUAL,eOperationModes.SEMI_AUTO:
			//direct changes
			currentMode := interfaceControl^.requestMode;
		eOperationModes.AUTO:
			//check : no error , manual channel work done
			IF errorDevice=0 THEN
				currentMode := eOperationModes.AUTO;
			ELSE
				//refuce to change , maintain
			END_IF 
	END_CASE
END_IF
//
CASE currentMode OF	
		eOperationModes.AUTO,eOperationModes.SEMI_AUTO:
		//running sequences
		FOR nCounter :=1 TO unitUpperBound BY 1 DO
			IF gvl.units[nCounter] <> 0 THEN
				gvl.units[nCounter]^();
			END_IF
		END_FOR
		
		IF  requestInitialize THEN
			//initialize all stations
			bAllInitialized := TRUE;
			interfaceControl^.state := TO_WORD(eSpecialStates.MAIN_INITIALIZING); //status reflection
			
			FOR nCounter:=1 TO unitUpperBound BY 1 DO
				IF gvl.units[nCounter] <> 0 THEN
					// if every station comes initialized
					bAllInitialized := bAllInitialized AND gvl.units[nCounter]^.Initialize();
				END_IF
			END_FOR
			IF bAllInitialized THEN
				FOR nCounter:=1 TO unitUpperBound BY 1 DO
					IF gvl.units[nCounter] <> 0 THEN
						gvl.units[nCounter]^.NextState := 0; //start working
					END_IF
				END_FOR	
				requestInitialize := FALSE; //clear after done
				//---------------------------------
				//	Clear all material valid status
				//---------------------------------
				FOR nCounter:=1 TO slotUpperBound BY 1 DO
					gvl.materialSlots[nCounter].Valid := FALSE;
				END_FOR
				
				interfaceControl^.state := TO_WORD(eSpecialStates.MAIN_INITIALIZED); //status reflection
			END_IF
		END_IF		
END_CASE

//status reflect
isInitializing := requestInitialize AND NOT bAllInitialized;
//

